C03591=1030.387,347.262,-133.744,171.985,46.375,159.086
C03592=1030.379,347.015,-133.707,171.979,46.373,159.085
C03593=1030.371,346.768,-133.670,171.972,46.372,159.084
C03594=1030.363,346.521,-133.633,171.966,46.372,159.083
C03595=1030.356,346.273,-133.596,171.960,46.371,159.082
C03596=1030.348,346.026,-133.559,171.954,46.370,159.081
C03597=1030.341,345.779,-133.521,171.948,46.368,159.080
C03598=1030.333,345.532,-133.484,171.942,46.367,159.079
C03599=1030.325,345.285,-133.447,171.936,46.366,159.078
C03600=1030.317,345.038,-133.410,171.930,46.365,159.077
C03601=1030.310,344.791,-133.372,171.924,46.364,159.076
C03602=1030.302,344.544,-133.336,171.918,46.363,159.075
C03603=1030.295,344.297,-133.298,171.912,46.362,159.074
C03604=1030.287,344.050,-133.262,171.906,46.361,159.073
C03605=1030.280,343.803,-133.224,171.899,46.360,159.072
C03606=1030.272,343.555,-133.188,171.894,46.359,159.072
C03607=1030.264,343.308,-133.151,171.887,46.358,159.071
C03608=1030.257,343.061,-133.113,171.881,46.357,159.070
C03609=1030.249,342.814,-133.077,171.875,46.356,159.069
C03610=1030.242,342.567,-133.040,171.869,46.355,159.068
C03611=1030.234,342.319,-133.003,171.864,46.354,159.067
C03612=1030.226,342.072,-132.966,171.858,46.353,159.066
C03613=1030.219,341.825,-132.929,171.852,46.352,159.065
C03614=1030.212,341.578,-132.893,171.846,46.351,159.064
C03615=1030.204,341.331,-132.855,171.840,46.350,159.063
C03616=1030.197,341.083,-132.819,171.833,46.349,159.062
C03617=1030.189,340.836,-132.783,171.828,46.349,159.061
C03618=1030.182,340.589,-132.746,171.822,46.347,159.060
C03619=1030.175,340.342,-132.709,171.816,46.347,159.060
C03620=1030.167,340.095,-132.672,171.810,46.346,159.059
C03621=1030.159,339.848,-132.636,171.804,46.345,159.058
C03622=1030.151,339.600,-132.600,171.798,46.344,159.057
C03623=1030.144,339.352,-132.563,171.792,46.343,159.056
C03624=1030.136,339.106,-132.526,171.787,46.343,159.055
C03625=1030.129,338.859,-132.490,171.781,46.341,159.054
C03626=1030.122,338.611,-132.454,171.775,46.341,159.053
C03627=1030.114,338.364,-132.418,171.769,46.340,159.053
C03628=1030.106,338.116,-132.382,171.763,46.339,159.052
C03629=1030.099,337.869,-132.346,171.758,46.338,159.051
C03630=1030.092,337.623,-132.308,171.752,46.338,159.050
C03631=1030.084,337.375,-132.272,171.746,46.337,159.049
C03632=1030.077,337.128,-132.236,171.740,46.336,159.048
C03633=1030.069,336.880,-132.200,171.734,46.336,159.047
C03634=1030.062,336.633,-132.164,171.729,46.335,159.047
C03635=1030.049,336.216,-132.102,171.720,46.334,159.045
C03636=1030.037,335.800,-132.042,171.710,46.332,159.044
C03637=1030.024,335.383,-131.981,171.701,46.331,159.042
C03638=1030.012,334.966,-131.920,171.691,46.330,159.041
C03639=1030.005,334.718,-131.884,171.685,46.330,159.040
C03640=1029.998,334.472,-131.848,171.679,46.328,159.039
C03641=1029.990,334.224,-131.812,171.674,46.328,159.038
C03642=1029.982,333.977,-131.776,171.668,46.327,159.038
C03643=1029.975,333.730,-131.740,171.662,46.326,159.037
C03644=1029.968,333.482,-131.704,171.656,46.326,159.036
C03645=1029.961,333.235,-131.669,171.652,46.326,159.035
C03646=1029.953,332.988,-131.632,171.646,46.325,159.034
C03647=1029.945,332.740,-131.597,171.640,46.325,159.034
C03648=1029.938,332.493,-131.562,171.635,46.324,159.033
C03649=1029.930,332.246,-131.525,171.629,46.323,159.032
C03650=1029.924,331.998,-131.490,171.623,46.323,159.031
C03651=1029.916,331.751,-131.454,171.617,46.322,159.030
C03652=1029.909,331.504,-131.419,171.612,46.321,159.030
C03653=1029.901,331.256,-131.383,171.606,46.321,159.029
C03654=1029.895,331.009,-131.347,171.601,46.321,159.028
C03655=1029.886,330.762,-131.312,171.596,46.320,159.027
C03656=1029.879,330.514,-131.277,171.590,46.319,159.027
C03657=1029.872,330.267,-131.241,171.584,46.319,159.026
C03658=1029.865,330.019,-131.205,171.579,46.319,159.025
C03659=1029.857,329.772,-131.169,171.574,46.318,159.024
C03660=1029.851,329.525,-131.134,171.569,46.317,159.024
C03661=1029.843,329.277,-131.098,171.563,46.317,159.023
C03662=1029.835,329.030,-131.063,171.557,46.317,159.022
C03663=1029.829,328.783,-131.028,171.552,46.316,159.021
C03664=1029.821,328.535,-130.992,171.546,46.315,159.021
C03665=1029.814,328.288,-130.957,171.541,46.316,159.020
C03666=1029.807,328.040,-130.921,171.536,46.315,159.019
C03667=1029.800,327.793,-130.885,171.530,46.314,159.018
C03668=1029.792,327.546,-130.851,171.525,46.314,159.018
C03669=1029.785,327.298,-130.815,171.519,46.313,159.017
C03670=1029.777,327.051,-130.781,171.514,46.313,159.016
C03671=1029.769,326.803,-130.746,171.509,46.313,159.015
C03672=1029.762,326.556,-130.711,171.503,46.313,159.015
C03673=1029.755,326.309,-130.676,171.498,46.313,159.014
C03674=1029.748,326.061,-130.641,171.493,46.312,159.013
C03675=1029.740,325.814,-130.606,171.487,46.312,159.013
C03676=1029.733,325.566,-130.571,171.482,46.311,159.012
C03677=1029.725,325.319,-130.536,171.477,46.311,159.011
C03678=1029.718,325.071,-130.502,171.471,46.311,159.011
C03679=1029.711,324.824,-130.467,171.466,46.310,159.010
C03680=1029.703,324.576,-130.432,171.460,46.310,159.009
C03681=1029.696,324.329,-130.396,171.456,46.310,159.009
C03682=1029.689,324.081,-130.363,171.450,46.310,159.008
C03683=1029.682,323.833,-130.327,171.444,46.310,159.007
C03684=1029.674,323.586,-130.293,171.440,46.310,159.007
C03685=1029.666,323.339,-130.258,171.434,46.310,159.006
C03686=1029.660,323.092,-130.223,171.429,46.309,159.005
C03687=1029.652,322.844,-130.188,171.424,46.309,159.005
C03688=1029.645,322.596,-130.154,171.419,46.309,159.004
C03689=1029.638,322.349,-130.119,171.413,46.309,159.003
C03690=1029.630,322.102,-130.085,171.408,46.308,159.003
C03691=1029.624,321.891,-130.054,171.404,46.308,159.002
C03692=1029.618,321.680,-130.026,171.399,46.308,159.002
C03693=1029.612,321.470,-129.996,171.395,46.308,159.001
C03694=1029.605,321.259,-129.967,171.390,46.308,159.000
C03695=1029.600,321.049,-129.937,171.386,46.307,159.000
C03696=1029.593,320.838,-129.907,171.381,46.307,158.999
C03697=1029.588,320.627,-129.878,171.377,46.307,158.999
C03698=1029.581,320.417,-129.849,171.373,46.307,158.998
C03699=1029.575,320.169,-129.814,171.367,46.307,158.998
C03700=1029.567,319.922,-129.780,171.363,46.306,158.997
C03701=1029.560,319.674,-129.745,171.357,46.306,158.996
C03702=1029.553,319.426,-129.711,171.352,46.306,158.996
C03703=1029.545,319.179,-129.676,171.347,46.306,158.995
C03704=1029.539,318.931,-129.642,171.342,46.306,158.994
C03705=1029.531,318.684,-129.607,171.337,46.306,158.994
C03706=1029.525,318.436,-129.573,171.332,46.306,158.993
C03707=1029.517,318.189,-129.538,171.327,46.306,158.993
C03708=1029.510,317.941,-129.505,171.322,46.306,158.992
C03709=1029.503,317.694,-129.469,171.317,46.305,158.991
C03710=1029.496,317.446,-129.436,171.311,46.305,158.991
C03711=1029.489,317.199,-129.401,171.307,46.305,158.990
C03712=1029.482,316.951,-129.367,171.301,46.305,158.989
C03713=1029.475,316.703,-129.333,171.297,46.305,158.989
C03714=1029.468,316.456,-129.298,171.291,46.305,158.988
C03715=1029.462,316.209,-129.264,171.286,46.305,158.988
C03716=1029.454,315.961,-129.230,171.282,46.305,158.987
C03717=1029.448,315.714,-129.195,171.276,46.305,158.987
C03718=1029.440,315.466,-129.161,171.272,46.305,158.986
C03719=1029.433,315.219,-129.128,171.266,46.305,158.985
C03720=1029.427,314.971,-129.093,171.262,46.305,158.985
C03721=1029.419,314.724,-129.059,171.257,46.305,158.984
C03722=1029.412,314.476,-129.025,171.251,46.305,158.984
C03723=1029.406,314.229,-128.991,171.247,46.305,158.983
C03724=1029.399,313.981,-128.957,171.241,46.305,158.982
C03725=1029.392,313.734,-128.922,171.237,46.305,158.982
C03726=1029.385,313.486,-128.888,171.232,46.305,158.981
C03727=1029.378,313.238,-128.854,171.227,46.305,158.981
C03728=1029.371,312.991,-128.820,171.222,46.305,158.980
C03729=1029.365,312.743,-128.786,171.218,46.305,158.980
C03730=1029.358,312.496,-128.752,171.212,46.305,158.979
C03731=1029.351,312.248,-128.718,171.207,46.305,158.978
C03732=1029.344,312.000,-128.684,171.203,46.305,158.978
C03733=1029.337,311.753,-128.651,171.197,46.305,158.977
C03734=1029.331,311.505,-128.616,171.193,46.305,158.977
C03735=1029.324,311.257,-128.583,171.188,46.305,158.976
C03736=1029.317,311.010,-128.549,171.183,46.306,158.976
C03737=1029.310,310.763,-128.515,171.178,46.305,158.975
C03738=1029.303,310.515,-128.481,171.174,46.306,158.975
C03739=1029.295,310.268,-128.448,171.168,46.306,158.974
C03740=1029.288,310.019,-128.415,171.164,46.306,158.974
C03741=1029.281,309.772,-128.382,171.158,46.306,158.973
C03742=1029.273,309.525,-128.348,171.154,46.307,158.973
C03743=1029.266,309.277,-128.315,171.149,46.306,158.972
C03744=1029.259,309.029,-128.281,171.144,46.307,158.972
C03745=1029.253,308.782,-128.248,171.140,46.307,158.971
C03746=1029.245,308.535,-128.215,171.134,46.307,158.970
C03747=1029.238,308.286,-128.182,171.130,46.308,158.970
C03748=1029.231,308.040,-128.148,171.126,46.308,158.970
C03749=1029.224,307.791,-128.115,171.120,46.308,158.969
C03750=1029.216,307.544,-128.082,171.116,46.309,158.969
C03751=1029.205,307.127,-128.026,171.108,46.309,158.968
C03752=1029.193,306.711,-127.970,171.099,46.309,158.967
C03753=1029.181,306.295,-127.914,171.091,46.310,158.966
C03754=1029.170,305.879,-127.859,171.084,46.311,158.965
C03755=1029.162,305.631,-127.825,171.079,46.311,158.965
C03756=1029.155,305.384,-127.793,171.074,46.312,158.964
C03757=1029.148,305.136,-127.759,171.069,46.311,158.964
C03758=1029.141,304.888,-127.726,171.065,46.312,158.963
C03759=1029.134,304.640,-127.694,171.060,46.312,158.963
C03760=1029.127,304.393,-127.660,171.055,46.313,158.963
C03761=1029.121,304.145,-127.627,171.051,46.313,158.962
C03762=1029.113,303.897,-127.595,171.046,46.313,158.961
C03763=1029.107,303.650,-127.561,171.041,46.314,158.961
C03764=1029.100,303.402,-127.528,171.037,46.314,158.961
C03765=1029.093,303.154,-127.495,171.033,46.314,158.960
C03766=1029.085,302.907,-127.462,171.027,46.315,158.960
C03767=1029.079,302.659,-127.429,171.023,46.316,158.959
C03768=1029.072,302.411,-127.396,171.019,46.316,158.959
C03769=1029.065,302.164,-127.364,171.014,46.316,158.958
C03770=1029.058,301.916,-127.330,171.009,46.316,158.958
C03771=1029.052,301.668,-127.298,171.004,46.317,158.957
C03772=1029.044,301.420,-127.265,171.000,46.317,158.957
C03773=1029.038,301.173,-127.232,170.996,46.318,158.957
C03774=1029.031,300.925,-127.199,170.990,46.318,158.956
C03775=1029.025,300.677,-127.166,170.986,46.319,158.956
C03776=1029.017,300.430,-127.133,170.982,46.319,158.955
C03777=1029.010,300.182,-127.100,170.977,46.319,158.955
C03778=1029.004,299.934,-127.068,170.973,46.320,158.954
C03779=1028.996,299.686,-127.035,170.968,46.320,158.954
C03780=1028.990,299.439,-127.002,170.963,46.321,158.954
C03781=1028.983,299.191,-126.969,170.959,46.321,158.953
C03782=1028.976,298.943,-126.937,170.955,46.322,158.953
C03783=1028.970,298.696,-126.904,170.950,46.322,158.952
C03784=1028.963,298.447,-126.871,170.945,46.323,158.952
C03785=1028.956,298.200,-126.839,170.941,46.323,158.951
C03786=1028.950,297.953,-126.806,170.936,46.323,158.951
C03787=1028.943,297.704,-126.773,170.932,46.324,158.951
C03788=1028.936,297.457,-126.741,170.928,46.324,158.950
C03789=1028.930,297.209,-126.708,170.922,46.325,158.950
C03790=1028.923,296.962,-126.676,170.918,46.325,158.949
C03791=1028.916,296.714,-126.643,170.914,46.326,158.949
C03792=1028.909,296.466,-126.610,170.909,46.326,158.948
C03793=1028.903,296.219,-126.578,170.905,46.327,158.948
C03794=1028.896,295.970,-126.546,170.901,46.328,158.948
C03795=1028.889,295.722,-126.513,170.897,46.328,158.947
C03796=1028.883,295.475,-126.480,170.891,46.329,158.947
C03797=1028.876,295.228,-126.448,170.887,46.329,158.946
C03798=1028.870,294.980,-126.416,170.883,46.329,158.946
C03799=1028.863,294.732,-126.382,170.878,46.330,158.946
C03800=1028.856,294.484,-126.351,170.874,46.331,158.945
C03801=1028.850,294.236,-126.318,170.870,46.331,158.945
C03802=1028.843,293.989,-126.286,170.866,46.332,158.945
C03803=1028.836,293.740,-126.254,170.860,46.332,158.944
C03804=1028.829,293.493,-126.222,170.856,46.333,158.944
C03805=1028.822,293.245,-126.189,170.852,46.334,158.943
C03806=1028.816,292.997,-126.157,170.848,46.334,158.943
C03807=1028.804,292.598,-126.106,170.840,46.335,158.942
C03808=1028.794,292.199,-126.054,170.834,46.336,158.942
C03809=1028.783,291.800,-126.002,170.827,46.337,158.941
C03810=1028.772,291.400,-125.951,170.820,46.339,158.941
C03811=1028.765,291.153,-125.919,170.815,46.339,158.940
C03812=1028.759,290.905,-125.887,170.811,46.340,158.940
C03813=1028.752,290.657,-125.855,170.807,46.341,158.940
C03814=1028.745,290.409,-125.824,170.803,46.341,158.939
C03815=1028.738,290.161,-125.792,170.799,46.342,158.939
C03816=1028.731,289.914,-125.760,170.793,46.343,158.939
C03817=1028.725,289.665,-125.728,170.789,46.344,158.938
C03818=1028.718,289.417,-125.696,170.785,46.344,158.938
C03819=1028.711,289.170,-125.664,170.781,46.345,158.938
C03820=1028.704,288.922,-125.633,170.777,46.346,158.938
C03821=1028.697,288.674,-125.601,170.772,46.347,158.937
C03822=1028.690,288.427,-125.569,170.768,46.348,158.937
C03823=1028.684,288.179,-125.537,170.764,46.348,158.936
C03824=1028.677,287.930,-125.505,170.759,46.350,158.936
C03825=1028.670,287.682,-125.474,170.755,46.350,158.936
C03826=1028.664,287.434,-125.442,170.751,46.351,158.935
C03827=1028.657,287.187,-125.410,170.747,46.352,158.935
C03828=1028.650,286.939,-125.379,170.742,46.352,158.935
C03829=1028.643,286.691,-125.347,170.738,46.353,158.935
C03830=1028.636,286.443,-125.316,170.734,46.354,158.934
C03831=1028.630,286.196,-125.284,170.730,46.355,158.934
C03832=1028.624,285.947,-125.252,170.726,46.356,158.934
C03833=1028.617,285.699,-125.221,170.722,46.357,158.933
C03834=1028.609,285.452,-125.190,170.717,46.357,158.933
C03835=1028.603,285.204,-125.159,170.712,46.359,158.933
C03836=1028.596,284.956,-125.127,170.708,46.360,158.932
C03837=1028.589,284.708,-125.096,170.704,46.361,158.932
C03838=1028.583,284.460,-125.064,170.700,46.361,158.932
C03839=1028.576,284.212,-125.033,170.696,46.362,158.932
C03840=1028.569,283.964,-125.001,170.692,46.363,158.931
C03841=1028.562,283.716,-124.970,170.688,46.364,158.931
C03842=1028.556,283.469,-124.939,170.684,46.365,158.931
C03843=1028.548,283.221,-124.908,170.680,46.366,158.931
C03844=1028.542,282.973,-124.876,170.676,46.367,158.930
C03845=1028.535,282.725,-124.846,170.671,46.368,158.930
C03846=1028.528,282.477,-124.814,170.667,46.369,158.930
C03847=1028.522,282.229,-124.783,170.663,46.370,158.929
C03848=1028.515,281.981,-124.751,170.658,46.371,158.929
C03849=1028.508,281.733,-124.720,170.654,46.372,158.929
C03850=1028.501,281.485,-124.688,170.650,46.373,158.929
C03851=1028.495,281.237,-124.658,170.646,46.373,158.928
C03852=1028.488,280.989,-124.627,170.642,46.374,158.928
C03853=1028.481,280.741,-124.595,170.638,46.375,158.928
C03854=1028.475,280.494,-124.564,170.634,46.376,158.927
C03855=1028.468,280.245,-124.534,170.630,46.377,158.927
C03856=1028.462,279.997,-124.502,170.626,46.378,158.927
C03857=1028.455,279.749,-124.471,170.622,46.379,158.927
C03858=1028.448,279.501,-124.440,170.618,46.381,158.926
C03859=1028.442,279.253,-124.409,170.614,46.382,158.926
C03860=1028.434,279.005,-124.378,170.610,46.383,158.926
C03861=1028.428,278.758,-124.347,170.606,46.384,158.926
C03862=1028.422,278.510,-124.316,170.601,46.385,158.925
C03863=1028.411,278.122,-124.267,170.595,46.386,158.925
C03864=1028.401,277.736,-124.219,170.589,46.388,158.925
C03865=1028.391,277.349,-124.171,170.582,46.389,158.924
C03866=1028.380,276.962,-124.122,170.576,46.391,158.924
C03867=1028.373,276.713,-124.092,170.572,46.392,158.924
C03868=1028.367,276.466,-124.062,170.568,46.393,158.923
C03869=1028.360,276.218,-124.031,170.564,46.394,158.923
C03870=1028.354,275.969,-124.000,170.560,46.396,158.923
C03871=1028.346,275.722,-123.969,170.556,46.397,158.923
C03872=1028.340,275.474,-123.939,170.552,46.398,158.923
C03873=1028.333,275.226,-123.908,170.548,46.399,158.922
C03874=1028.327,274.978,-123.877,170.544,46.400,158.922
C03875=1028.320,274.729,-123.846,170.540,46.401,158.922
C03876=1028.313,274.482,-123.815,170.536,46.403,158.922
C03877=1028.307,274.234,-123.785,170.532,46.404,158.922
C03878=1028.300,273.985,-123.754,170.528,46.405,158.921
C03879=1028.293,273.737,-123.724,170.524,46.406,158.921
C03880=1028.287,273.490,-123.693,170.520,46.407,158.921
C03881=1028.280,273.242,-123.663,170.516,46.408,158.921
C03882=1028.274,272.993,-123.632,170.512,46.409,158.921
C03883=1028.266,272.745,-123.602,170.508,46.410,158.920
C03884=1028.260,272.498,-123.571,170.504,46.411,158.920
C03885=1028.254,272.249,-123.540,170.501,46.413,158.920
C03886=1028.247,272.001,-123.510,170.497,46.414,158.920
C03887=1028.241,271.753,-123.480,170.493,46.415,158.919
C03888=1028.234,271.505,-123.450,170.489,46.417,158.919
C03889=1028.227,271.257,-123.418,170.485,46.418,158.919
C03890=1028.220,271.009,-123.389,170.481,46.419,158.919
C03891=1028.214,270.761,-123.358,170.477,46.421,158.919
C03892=1028.207,270.513,-123.328,170.474,46.421,158.919
C03893=1028.201,270.265,-123.298,170.470,46.422,158.918
C03894=1028.194,270.017,-123.267,170.466,46.424,158.918
C03895=1028.187,269.768,-123.237,170.462,46.425,158.918
C03896=1028.181,269.521,-123.207,170.458,46.427,158.918
C03897=1028.174,269.272,-123.177,170.454,46.428,158.918
C03898=1028.167,269.024,-123.146,170.450,46.429,158.917
C03899=1028.161,268.776,-123.116,170.446,46.430,158.917
C03900=1028.154,268.528,-123.086,170.442,46.431,158.917
C03901=1028.148,268.280,-123.056,170.439,46.433,158.917
C03902=1028.141,268.032,-123.026,170.435,46.434,158.917
C03903=1028.133,267.784,-122.996,170.431,46.436,158.917
C03904=1028.128,267.536,-122.965,170.427,46.437,158.916
C03905=1028.121,267.288,-122.935,170.423,46.438,158.916
C03906=1028.114,267.040,-122.905,170.419,46.440,158.916
C03907=1028.108,266.791,-122.875,170.415,46.441,158.916
C03908=1028.101,266.544,-122.846,170.411,46.442,158.916
C03909=1028.094,266.296,-122.816,170.407,46.444,158.916
C03910=1028.088,266.047,-122.785,170.403,46.445,158.916
C03911=1028.081,265.799,-122.755,170.401,46.446,158.916
C03912=1028.074,265.551,-122.726,170.397,46.447,158.915
C03913=1028.068,265.303,-122.696,170.393,46.449,158.915
C03914=1028.061,265.055,-122.665,170.389,46.451,158.915
C03915=1028.055,264.807,-122.635,170.385,46.452,158.915
C03916=1028.048,264.558,-122.606,170.381,46.453,158.915
C03917=1028.041,264.311,-122.576,170.377,46.454,158.915
C03918=1028.034,264.063,-122.546,170.374,46.456,158.914
C03919=1028.024,263.680,-122.500,170.368,46.458,158.914
C03920=1028.014,263.298,-122.454,170.362,46.460,158.914
C03921=1028.004,262.915,-122.408,170.356,46.463,158.914
C03922=1027.994,262.533,-122.363,170.350,46.465,158.914
C03923=1027.987,262.285,-122.332,170.347,46.466,158.914
C03924=1027.981,262.037,-122.303,170.343,46.467,158.913
C03925=1027.974,261.788,-122.273,170.339,46.469,158.913
C03926=1027.968,261.540,-122.244,170.335,46.471,158.913
C03927=1027.961,261.293,-122.214,170.331,46.472,158.913
C03928=1027.954,261.044,-122.184,170.328,46.473,158.913
C03929=1027.948,260.796,-122.155,170.325,46.475,158.913
C03930=1027.941,260.548,-122.126,170.321,46.477,158.913
C03931=1027.934,260.300,-122.096,170.317,46.478,158.913
C03932=1027.927,260.051,-122.066,170.313,46.480,158.913
C03933=1027.921,259.804,-122.037,170.310,46.482,158.912
C03934=1027.913,259.555,-122.008,170.306,46.483,158.912
C03935=1027.907,259.307,-121.979,170.302,46.484,158.912
C03936=1027.900,259.059,-121.949,170.298,46.486,158.912
C03937=1027.894,258.811,-121.920,170.294,46.488,158.912
C03938=1027.887,258.563,-121.891,170.291,46.489,158.912
C03939=1027.880,258.314,-121.862,170.287,46.491,158.912
C03940=1027.873,258.067,-121.832,170.283,46.493,158.912
C03941=1027.866,257.818,-121.803,170.279,46.494,158.912
C03942=1027.860,257.570,-121.774,170.277,46.496,158.912
C03943=1027.853,257.321,-121.744,170.273,46.497,158.912
C03944=1027.846,257.074,-121.715,170.269,46.499,158.912
C03945=1027.840,256.825,-121.686,170.265,46.501,158.911
C03946=1027.833,256.577,-121.657,170.262,46.502,158.911
C03947=1027.827,256.328,-121.627,170.258,46.504,158.911
C03948=1027.820,256.081,-121.599,170.254,46.506,158.911
C03949=1027.812,255.832,-121.569,170.250,46.507,158.911
C03950=1027.806,255.584,-121.540,170.247,46.509,158.911
C03951=1027.799,255.335,-121.510,170.243,46.511,158.911
C03952=1027.793,255.087,-121.481,170.240,46.512,158.911
C03953=1027.786,254.839,-121.453,170.236,46.514,158.911
C03954=1027.779,254.591,-121.424,170.233,46.516,158.911
C03955=1027.773,254.342,-121.395,170.229,46.517,158.911
C03956=1027.767,254.094,-121.365,170.225,46.519,158.911
C03957=1027.760,253.847,-121.337,170.221,46.521,158.911
C03958=1027.753,253.598,-121.307,170.217,46.522,158.910
C03959=1027.746,253.350,-121.278,170.214,46.524,158.910
C03960=1027.740,253.102,-121.249,170.211,46.525,158.910
C03961=1027.733,252.853,-121.219,170.207,46.527,158.910
C03962=1027.726,252.605,-121.191,170.203,46.529,158.910
C03963=1027.720,252.357,-121.162,170.200,46.530,158.910
C03964=1027.714,252.109,-121.133,170.196,46.532,158.910
C03965=1027.707,251.860,-121.103,170.192,46.534,158.910
C03966=1027.700,251.612,-121.075,170.188,46.535,158.910
C03967=1027.694,251.364,-121.046,170.186,46.537,158.910
C03968=1027.687,251.116,-121.017,170.182,46.539,158.910
C03969=1027.681,250.867,-120.988,170.179,46.541,158.910
C03970=1027.674,250.620,-120.959,170.175,46.542,158.910
C03971=1027.668,250.371,-120.931,170.171,46.544,158.910
C03972=1027.661,250.123,-120.902,170.167,46.546,158.910
C03973=1027.655,249.875,-120.873,170.164,46.547,158.910
C03974=1027.648,249.626,-120.844,170.161,46.549,158.909
C03975=1027.638,249.242,-120.799,170.155,46.552,158.909
C03976=1027.628,248.859,-120.754,170.150,46.555,158.909
C03977=1027.618,248.475,-120.710,170.144,46.557,158.909
C03978=1027.608,248.091,-120.665,170.139,46.560,158.909
C03979=1027.601,247.843,-120.636,170.135,46.562,158.909
C03980=1027.595,247.594,-120.608,170.132,46.563,158.909
C03981=1027.589,247.346,-120.579,170.129,46.565,158.909
C03982=1027.583,247.098,-120.550,170.125,46.567,158.909
C03983=1027.576,246.850,-120.522,170.121,46.569,158.909
C03984=1027.569,246.601,-120.492,170.118,46.571,158.909
C03985=1027.563,246.353,-120.464,170.115,46.572,158.909
C03986=1027.557,246.105,-120.435,170.111,46.574,158.909
C03987=1027.550,245.857,-120.406,170.107,46.575,158.909
C03988=1027.543,245.609,-120.377,170.104,46.578,158.909
C03989=1027.537,245.360,-120.349,170.101,46.579,158.909
C03990=1027.531,245.112,-120.320,170.097,46.581,158.909
C03991=1027.524,244.864,-120.291,170.094,46.583,158.909
C03992=1027.518,244.615,-120.263,170.090,46.585,158.909
C03993=1027.512,244.367,-120.234,170.086,46.587,158.909
C03994=1027.505,244.119,-120.206,170.084,46.588,158.909
C03995=1027.499,243.870,-120.177,170.080,46.590,158.909
C03996=1027.492,243.623,-120.149,170.076,46.592,158.909
C03997=1027.486,243.374,-120.121,170.073,46.594,158.909
C03998=1027.479,243.125,-120.092,170.069,46.596,158.909
C03999=1027.473,242.877,-120.063,170.066,46.597,158.909
C04000=1027.466,242.629,-120.035,170.063,46.599,158.909
C04001=1027.460,242.380,-120.007,170.059,46.601,158.909
C04002=1027.453,242.132,-119.978,170.055,46.603,158.909
C04003=1027.447,241.883,-119.950,170.053,46.605,158.909
C04004=1027.440,241.636,-119.921,170.049,46.607,158.909
C04005=1027.434,241.387,-119.893,170.046,46.609,158.909
C04006=1027.427,241.139,-119.865,170.042,46.611,158.909
C04007=1027.420,240.891,-119.837,170.038,46.613,158.909
C04008=1027.414,240.642,-119.808,170.036,46.615,158.909
C04009=1027.407,240.394,-119.780,170.032,46.616,158.909
C04010=1027.401,240.145,-119.752,170.029,46.619,158.909
C04011=1027.394,239.897,-119.723,170.025,46.620,158.909
C04012=1027.388,239.649,-119.696,170.021,46.623,158.909
C04013=1027.382,239.400,-119.667,170.019,46.624,158.909
C04014=1027.375,239.152,-119.639,170.015,46.626,158.909
C04015=1027.368,238.904,-119.611,170.011,46.628,158.909
C04016=1027.361,238.656,-119.583,170.008,46.630,158.909
C04017=1027.355,238.407,-119.556,170.005,46.633,158.909
C04018=1027.348,238.159,-119.527,170.002,46.634,158.909
C04019=1027.342,237.911,-119.499,169.998,46.636,158.909
C04020=1027.335,237.662,-119.471,169.995,46.638,158.909
C04021=1027.328,237.414,-119.443,169.991,46.641,158.909
C04022=1027.322,237.165,-119.416,169.988,46.643,158.909
C04023=1027.315,236.917,-119.387,169.985,46.644,158.909
C04024=1027.309,236.669,-119.359,169.981,46.647,158.909
C04025=1027.302,236.420,-119.331,169.978,46.649,158.909
C04026=1027.295,236.172,-119.304,169.974,46.651,158.909
C04027=1027.289,235.924,-119.276,169.971,46.653,158.909
C04028=1027.283,235.676,-119.248,169.968,46.655,158.909
C04029=1027.276,235.427,-119.221,169.965,46.657,158.909
C04030=1027.270,235.178,-119.192,169.961,46.659,158.909
C04031=1027.259,234.789,-119.149,169.956,46.663,158.909
C04032=1027.249,234.398,-119.104,169.950,46.665,158.909
C04033=1027.239,234.009,-119.061,169.945,46.669,158.910
C04034=1027.229,233.619,-119.018,169.940,46.672,158.910
C04035=1027.222,233.370,-118.990,169.937,46.674,158.910
C04036=1027.215,233.122,-118.962,169.934,46.676,158.910
C04037=1027.209,232.873,-118.934,169.930,46.678,158.910
C04038=1027.202,232.625,-118.907,169.927,46.681,158.910
C04039=1027.196,232.377,-118.879,169.924,46.682,158.910
C04040=1027.189,232.129,-118.852,169.921,46.685,158.910
C04041=1027.183,231.880,-118.824,169.917,46.687,158.910
C04042=1027.177,231.631,-118.795,169.914,46.689,158.910
C04043=1027.170,231.383,-118.768,169.911,46.691,158.910
C04044=1027.163,231.135,-118.740,169.908,46.693,158.910
C04045=1027.157,230.887,-118.713,169.904,46.695,158.910
C04046=1027.150,230.638,-118.685,169.901,46.698,158.910
C04047=1027.144,230.390,-118.657,169.898,46.700,158.911
C04048=1027.137,230.141,-118.630,169.894,46.701,158.910
C04049=1027.131,229.892,-118.602,169.891,46.704,158.911
C04050=1027.124,229.644,-118.575,169.888,46.706,158.911
C04051=1027.118,229.396,-118.547,169.885,46.708,158.911
C04052=1027.111,229.148,-118.520,169.882,46.711,158.911
C04053=1027.105,228.899,-118.492,169.878,46.713,158.911
C04054=1027.098,228.650,-118.465,169.875,46.715,158.911
C04055=1027.092,228.402,-118.437,169.872,46.717,158.911
C04056=1027.085,228.154,-118.410,169.869,46.719,158.911
C04057=1027.079,227.906,-118.382,169.865,46.721,158.911
C04058=1027.072,227.657,-118.356,169.862,46.724,158.911
C04059=1027.065,227.408,-118.328,169.859,46.726,158.911
C04060=1027.059,227.161,-118.301,169.856,46.728,158.911
C04061=1027.053,226.912,-118.274,169.852,46.730,158.912
C04062=1027.046,226.663,-118.246,169.849,46.733,158.912
C04063=1027.038,226.415,-118.219,169.846,46.735,158.912
C04064=1027.033,226.167,-118.192,169.843,46.737,158.912
C04065=1027.026,225.918,-118.164,169.839,46.740,158.912
C04066=1027.020,225.669,-118.137,169.836,46.742,158.912
C04067=1027.012,225.421,-118.110,169.832,46.744,158.912
C04068=1027.006,225.173,-118.082,169.830,46.746,158.912
C04069=1027.000,224.924,-118.056,169.827,46.749,158.912
C04070=1026.992,224.676,-118.029,169.823,46.751,158.912
C04071=1026.986,224.427,-118.002,169.820,46.753,158.912
C04072=1026.980,224.179,-117.974,169.817,46.755,158.913
C04073=1026.974,223.930,-117.947,169.814,46.758,158.913
C04074=1026.966,223.682,-117.920,169.811,46.761,158.913
C04075=1026.960,223.433,-117.893,169.807,46.763,158.913
C04076=1026.954,223.185,-117.866,169.805,46.765,158.913
C04077=1026.947,222.937,-117.839,169.801,46.768,158.913
C04078=1026.940,222.688,-117.812,169.798,46.770,158.913
C04079=1026.934,222.440,-117.785,169.794,46.772,158.913
C04080=1026.927,222.191,-117.757,169.792,46.774,158.914
C04081=1026.920,221.943,-117.731,169.788,46.777,158.914
C04082=1026.914,221.695,-117.703,169.785,46.779,158.914
C04083=1026.908,221.446,-117.676,169.782,46.781,158.914
C04084=1026.901,221.197,-117.650,169.779,46.784,158.914
C04085=1026.895,220.949,-117.623,169.776,46.786,158.914
C04086=1026.888,220.700,-117.596,169.772,46.789,158.914
C04087=1026.877,220.303,-117.552,169.767,46.792,158.914
C04088=1026.868,219.905,-117.509,169.762,46.796,158.915
C04089=1026.857,219.508,-117.466,169.758,46.800,158.915
C04090=1026.847,219.110,-117.423,169.753,46.803,158.915
C04091=1026.840,218.861,-117.396,169.750,46.806,158.915
C04092=1026.833,218.613,-117.369,169.746,46.809,158.915
C04093=1026.826,218.365,-117.343,169.743,46.811,158.915
C04094=1026.820,218.116,-117.316,169.741,46.814,158.916
C04095=1026.813,217.868,-117.289,169.737,46.816,158.916
C04096=1026.807,217.619,-117.262,169.734,46.818,158.916
C04097=1026.800,217.370,-117.236,169.730,46.821,158.916
C04098=1026.794,217.122,-117.209,169.728,46.823,158.916
C04099=1026.787,216.873,-117.183,169.725,46.826,158.916
C04100=1026.780,216.625,-117.157,169.721,46.828,158.916
C04101=1026.774,216.377,-117.129,169.718,46.831,158.917
C04102=1026.767,216.128,-117.103,169.716,46.833,158.917
C04103=1026.761,215.880,-117.076,169.712,46.836,158.917
C04104=1026.754,215.631,-117.050,169.709,46.839,158.917
C04105=1026.748,215.382,-117.023,169.706,46.841,158.917
C04106=1026.741,215.134,-116.996,169.703,46.843,158.917
C04107=1026.734,214.886,-116.970,169.700,46.846,158.918
C04108=1026.728,214.637,-116.943,169.697,46.848,158.918
C04109=1026.721,214.388,-116.917,169.693,46.851,158.918
C04110=1026.715,214.140,-116.890,169.691,46.853,158.918
C04111=1026.708,213.891,-116.863,169.687,46.856,158.918
C04112=1026.701,213.643,-116.837,169.684,46.859,158.918
C04113=1026.695,213.394,-116.810,169.682,46.861,158.919
C04114=1026.688,213.146,-116.784,169.678,46.863,158.919
C04115=1026.682,212.897,-116.757,169.675,46.866,158.919
C04116=1026.675,212.649,-116.731,169.672,46.869,158.919
C04117=1026.669,212.400,-116.704,169.669,46.871,158.919
C04118=1026.662,212.152,-116.678,169.666,46.874,158.919
C04119=1026.655,211.903,-116.652,169.663,46.876,158.919
C04120=1026.650,211.655,-116.625,169.661,46.879,158.920
C04121=1026.642,211.406,-116.598,169.657,46.881,158.920
C04122=1026.637,211.158,-116.572,169.654,46.884,158.920
C04123=1026.630,210.909,-116.545,169.651,46.886,158.920
C04124=1026.623,210.661,-116.519,169.648,46.889,158.920
C04125=1026.617,210.412,-116.492,169.645,46.892,158.921
C04126=1026.610,210.163,-116.467,169.641,46.894,158.921
C04127=1026.604,209.915,-116.441,169.639,46.897,158.921
C04128=1026.597,209.666,-116.415,169.636,46.899,158.921
C04129=1026.590,209.418,-116.388,169.633,46.902,158.921
C04130=1026.584,209.169,-116.361,169.629,46.905,158.921
C04131=1026.577,208.921,-116.335,169.627,46.907,158.922
C04132=1026.570,208.673,-116.309,169.624,46.910,158.922
C04133=1026.564,208.424,-116.284,169.620,46.913,158.922
C04134=1026.558,208.175,-116.257,169.618,46.915,158.922
C04135=1026.551,207.927,-116.231,169.615,46.918,158.922
C04136=1026.544,207.678,-116.204,169.612,46.921,158.923
C04137=1026.538,207.429,-116.179,169.608,46.923,158.923
C04138=1026.531,207.181,-116.153,169.606,46.926,158.923
C04139=1026.524,206.933,-116.126,169.603,46.928,158.923
C04140=1026.518,206.685,-116.100,169.599,46.931,158.923
C04141=1026.512,206.435,-116.074,169.597,46.934,158.924
C04142=1026.505,206.187,-116.048,169.594,46.936,158.924
C04143=1026.494,205.793,-116.006,169.589,46.941,158.924
C04144=1026.484,205.399,-115.966,169.584,46.945,158.924
C04145=1026.474,205.006,-115.924,169.580,46.950,158.925
C04146=1026.463,204.611,-115.884,169.575,46.954,158.925
C04147=1026.439,203.573,-115.781,169.186,46.851,158.855
C04148=1026.432,203.324,-115.756,169.182,46.855,158.856
C04149=1026.427,203.076,-115.732,169.178,46.858,158.856
C04150=1026.421,202.827,-115.708,169.174,46.862,158.856
C04151=1026.415,202.578,-115.683,169.170,46.865,158.856
C04152=1026.409,202.329,-115.658,169.166,46.869,158.857
C04153=1026.403,202.081,-115.634,169.162,46.873,158.857
C04154=1026.397,201.832,-115.610,169.158,46.876,158.857
C04155=1026.392,201.583,-115.585,169.155,46.880,158.857
C04156=1026.386,201.334,-115.561,169.151,46.883,158.858
C04157=1026.381,201.086,-115.536,169.147,46.887,158.858
C04158=1026.375,200.838,-115.512,169.143,46.890,158.858
C04159=1026.369,200.588,-115.488,169.139,46.894,158.858
C04160=1026.363,200.340,-115.463,169.135,46.897,158.859
C04161=1026.357,200.090,-115.439,169.131,46.901,158.859
C04162=1026.351,199.842,-115.415,169.127,46.904,158.859
C04163=1026.345,199.593,-115.390,169.124,46.908,158.859
C04164=1026.339,199.345,-115.367,169.119,46.912,158.860
C04165=1026.334,199.095,-115.342,169.116,46.915,158.860
C04166=1026.328,198.847,-115.318,169.112,46.919,158.860
C04167=1026.321,198.598,-115.294,169.107,46.923,158.860
C04168=1026.316,198.350,-115.270,169.104,46.927,158.861
C04169=1026.309,198.101,-115.246,169.100,46.931,158.861
C04170=1026.304,197.851,-115.223,169.095,46.934,158.861
C04171=1026.298,197.603,-115.199,169.092,46.938,158.862
C04172=1026.292,197.354,-115.174,169.089,46.942,158.862
C04173=1026.286,197.105,-115.151,169.084,46.945,158.862
C04174=1026.279,196.856,-115.127,169.081,46.949,158.862
C04175=1026.274,196.608,-115.102,169.077,46.953,158.863
C04176=1026.268,196.360,-115.079,169.072,46.956,158.863
C04177=1026.262,196.110,-115.055,169.069,46.960,158.863
C04178=1026.256,195.861,-115.031,169.065,46.964,158.864
C04179=1026.251,195.613,-115.007,169.062,46.967,158.864
C04180=1026.244,195.364,-114.983,169.058,46.971,158.864
C04181=1026.238,195.116,-114.959,169.054,46.975,158.864
C04182=1026.233,194.866,-114.936,169.050,46.978,158.865
C04183=1026.227,194.617,-114.912,169.046,46.982,158.865
C04184=1026.221,194.369,-114.887,169.042,46.986,158.865
C04185=1026.215,194.121,-114.864,169.039,46.989,158.865
C04186=1026.209,193.871,-114.840,169.035,46.993,158.866
C04187=1026.204,193.622,-114.816,169.031,46.997,158.866
C04188=1026.198,193.374,-114.792,169.027,47.000,158.866
C04189=1026.192,193.124,-114.769,169.023,47.004,158.867
C04190=1026.186,192.876,-114.745,169.019,47.008,158.867
C04191=1026.181,192.627,-114.721,169.016,47.012,158.867
C04192=1026.175,192.379,-114.697,169.012,47.015,158.867
C04193=1026.168,192.129,-114.674,169.008,47.019,158.868
C04194=1026.163,191.881,-114.649,169.004,47.023,158.868
C04195=1026.157,191.632,-114.626,169.001,47.026,158.868
C04196=1026.152,191.383,-114.602,168.997,47.030,158.869
C04197=1026.145,191.134,-114.578,168.993,47.034,158.869
C04198=1026.140,190.885,-114.555,168.989,47.038,158.869
C04199=1026.134,190.637,-114.531,168.986,47.041,158.870
C04200=1026.129,190.388,-114.508,168.982,47.045,158.870
C04201=1026.123,190.139,-114.483,168.978,47.049,158.870
C04202=1026.117,189.890,-114.460,168.974,47.053,158.871
C04203=1026.111,189.642,-114.437,168.971,47.056,158.871
C04204=1026.106,189.393,-114.413,168.967,47.060,158.871
C04205=1026.100,189.144,-114.390,168.963,47.064,158.871
C04206=1026.094,188.895,-114.365,168.960,47.068,158.872
C04207=1026.088,188.646,-114.342,168.956,47.071,158.872
C04208=1026.083,188.410,-114.319,168.952,47.075,158.872
C04209=1026.078,188.174,-114.297,168.949,47.078,158.872
C04210=1026.072,187.938,-114.275,168.945,47.082,158.873
C04211=1026.066,187.702,-114.253,168.943,47.086,158.873
C04212=1026.061,187.466,-114.230,168.938,47.089,158.873
C04213=1026.056,187.231,-114.208,168.935,47.093,158.874
C04214=1026.051,186.994,-114.185,168.931,47.096,158.874
C04215=1026.046,186.758,-114.163,168.928,47.100,158.874
C04216=1026.040,186.509,-114.140,168.925,47.104,158.875
C04217=1026.034,186.260,-114.117,168.921,47.107,158.875
C04218=1026.028,186.011,-114.092,168.917,47.111,158.875
C04219=1026.022,185.762,-114.069,168.914,47.115,158.875
C04220=1026.017,185.514,-114.045,168.911,47.118,158.876
C04221=1026.011,185.265,-114.022,168.907,47.122,158.876
C04222=1026.006,185.016,-113.999,168.903,47.126,158.876
C04223=1026.000,184.767,-113.975,168.900,47.129,158.877
C04224=1025.995,184.518,-113.952,168.896,47.133,158.877
C04225=1025.989,184.269,-113.929,168.892,47.137,158.877
C04226=1025.984,184.021,-113.905,168.889,47.140,158.878
C04227=1025.978,183.772,-113.882,168.885,47.144,158.878
C04228=1025.973,183.523,-113.858,168.881,47.148,158.878
C04229=1025.967,183.274,-113.835,168.878,47.152,158.879
C04230=1025.961,183.026,-113.812,168.874,47.155,158.879
C04231=1025.956,182.776,-113.788,168.871,47.159,158.879
C04232=1025.950,182.527,-113.765,168.867,47.163,158.879
C04233=1025.944,182.278,-113.742,168.863,47.167,158.880
C04234=1025.938,182.029,-113.719,168.860,47.171,158.880
C04235=1025.932,181.781,-113.696,168.857,47.175,158.881
C04236=1025.926,181.532,-113.673,168.853,47.179,158.881
C04237=1025.920,181.283,-113.650,168.849,47.183,158.881
C04238=1025.914,181.035,-113.628,168.845,47.187,158.882
C04239=1025.908,180.785,-113.605,168.842,47.191,158.882
C04240=1025.902,180.536,-113.582,168.839,47.195,158.882
C04241=1025.897,180.287,-113.559,168.835,47.199,158.883
C04242=1025.890,180.039,-113.537,168.832,47.203,158.883
C04243=1025.885,179.790,-113.514,168.828,47.207,158.883
C04244=1025.877,179.481,-113.485,168.823,47.212,158.884
C04245=1025.870,179.173,-113.457,168.819,47.217,158.884
C04246=1025.862,178.865,-113.429,168.815,47.222,158.885
C04247=1025.855,178.556,-113.401,168.811,47.227,158.885
C04248=1025.849,178.308,-113.378,168.807,47.231,158.886
C04249=1025.844,178.059,-113.355,168.803,47.235,158.886
C04250=1025.837,177.810,-113.333,168.800,47.239,158.886
C04251=1025.832,177.561,-113.311,168.796,47.243,158.887
C04252=1025.826,177.312,-113.288,168.793,47.247,158.887
C04253=1025.820,177.063,-113.265,168.790,47.250,158.887
C04254=1025.814,176.814,-113.242,168.786,47.255,158.888
C04255=1025.808,176.565,-113.219,168.782,47.259,158.888
C04256=1025.802,176.316,-113.196,168.779,47.263,158.888
C04257=1025.797,176.067,-113.174,168.776,47.267,158.889
C04258=1025.791,175.818,-113.152,168.772,47.271,158.889
C04259=1025.785,175.569,-113.129,168.769,47.275,158.890
C04260=1025.779,175.320,-113.106,168.765,47.279,158.890
C04261=1025.773,175.072,-113.084,168.761,47.283,158.890
C04262=1025.767,174.822,-113.061,168.758,47.287,158.891
C04263=1025.761,174.573,-113.038,168.755,47.291,158.891
C04264=1025.756,174.325,-113.016,168.752,47.295,158.891
C04265=1025.750,174.076,-112.994,168.748,47.299,158.892
C04266=1025.744,173.827,-112.971,168.744,47.303,158.892
C04267=1025.739,173.578,-112.948,168.741,47.306,158.892
C04268=1025.733,173.329,-112.925,168.737,47.310,158.893
C04269=1025.727,173.080,-112.904,168.734,47.315,158.893
C04270=1025.721,172.831,-112.881,168.731,47.319,158.894
C04271=1025.715,172.582,-112.858,168.727,47.323,158.894
C04272=1025.709,172.299,-112.833,168.723,47.328,158.894
C04273=1025.702,172.017,-112.807,168.720,47.332,158.895
C04274=1025.696,171.733,-112.781,168.716,47.336,158.895
C04275=1025.689,171.450,-112.756,168.711,47.341,158.896
C04276=1025.684,171.201,-112.733,168.709,47.345,158.896
C04277=1025.678,170.952,-112.712,168.705,47.349,158.896
C04278=1025.672,170.703,-112.689,168.702,47.353,158.897
C04279=1025.667,170.454,-112.666,168.698,47.357,158.897
C04280=1025.660,170.205,-112.644,168.695,47.361,158.898
C04281=1025.655,169.956,-112.621,168.692,47.365,158.898
C04282=1025.649,169.707,-112.599,168.689,47.369,158.898
C04283=1025.644,169.458,-112.576,168.685,47.373,158.899
C04284=1025.638,169.210,-112.554,168.681,47.377,158.899
C04285=1025.632,168.961,-112.532,168.678,47.381,158.899
C04286=1025.627,168.712,-112.509,168.674,47.385,158.900
C04287=1025.620,168.462,-112.487,168.672,47.389,158.900
C04288=1025.615,168.214,-112.465,168.668,47.393,158.900
C04289=1025.610,167.965,-112.443,168.665,47.397,158.901
C04290=1025.604,167.716,-112.420,168.661,47.401,158.901
C04291=1025.598,167.467,-112.398,168.658,47.405,158.902
C04292=1025.593,167.218,-112.376,168.654,47.409,158.902
C04293=1025.587,166.969,-112.353,168.652,47.413,158.902
C04294=1025.581,166.720,-112.331,168.648,47.417,158.903
C04295=1025.576,166.471,-112.309,168.645,47.421,158.903
C04296=1025.570,166.223,-112.286,168.641,47.425,158.903
C04297=1025.564,165.973,-112.264,168.638,47.429,158.904
C04298=1025.559,165.724,-112.242,168.635,47.433,158.904
C04299=1025.554,165.476,-112.220,168.632,47.436,158.904
C04300=1025.548,165.227,-112.198,168.628,47.441,158.905
C04301=1025.542,164.978,-112.175,168.625,47.445,158.905
C04302=1025.537,164.729,-112.153,168.621,47.449,158.906
C04303=1025.532,164.479,-112.131,168.619,47.453,158.906
C04304=1025.525,164.231,-112.109,168.616,47.456,158.906
C04305=1025.520,163.982,-112.087,168.612,47.460,158.907
C04306=1025.515,163.733,-112.064,168.609,47.465,158.907
C04307=1025.508,163.484,-112.042,168.606,47.469,158.908
C04308=1025.504,163.235,-112.020,168.603,47.473,158.908
C04309=1025.498,162.986,-111.997,168.599,47.477,158.908
C04310=1025.492,162.737,-111.976,168.596,47.480,158.909
C04311=1025.487,162.488,-111.954,168.592,47.484,158.909
C04312=1025.481,162.239,-111.931,168.589,47.488,158.909
C04313=1025.475,161.990,-111.909,168.587,47.493,158.910
C04314=1025.470,161.741,-111.887,168.583,47.497,158.910
C04315=1025.464,161.492,-111.864,168.580,47.500,158.911
C04316=1025.459,161.244,-111.843,168.576,47.504,158.911
C04317=1025.453,160.994,-111.821,168.573,47.508,158.911
C04318=1025.448,160.745,-111.799,168.570,47.512,158.912
C04319=1025.442,160.497,-111.777,168.567,47.517,158.912
C04320=1025.437,160.247,-111.755,168.564,47.520,158.912
C04321=1025.432,159.998,-111.733,168.560,47.525,158.913
C04322=1025.426,159.749,-111.711,168.557,47.528,158.913
C04323=1025.421,159.501,-111.688,168.555,47.532,158.914
C04324=1025.415,159.252,-111.666,168.551,47.536,158.914
C04325=1025.409,159.002,-111.645,168.548,47.541,158.914
C04326=1025.403,158.754,-111.623,168.544,47.545,158.915
C04327=1025.397,158.505,-111.602,168.541,47.548,158.915
C04328=1025.392,158.255,-111.579,168.538,47.553,158.916
C04329=1025.386,158.007,-111.558,168.535,47.557,158.916
C04330=1025.380,157.757,-111.537,168.532,47.562,158.916
C04331=1025.375,157.509,-111.515,168.529,47.565,158.917
C04332=1025.369,157.259,-111.493,168.525,47.569,158.917
C04333=1025.363,157.010,-111.471,168.522,47.574,158.918
C04334=1025.357,156.762,-111.450,168.519,47.578,158.918
C04335=1025.351,156.512,-111.429,168.516,47.582,158.919
C04336=1025.346,156.229,-111.404,168.512,47.587,158.919
C04337=1025.339,155.945,-111.380,168.509,47.592,158.919
C04338=1025.332,155.662,-111.355,168.505,47.596,158.920
C04339=1025.326,155.378,-111.330,168.502,47.601,158.920
C04340=1025.320,155.129,-111.309,168.498,47.605,158.921
C04341=1025.314,154.880,-111.287,168.495,47.609,158.921
C04342=1025.309,154.631,-111.266,168.493,47.613,158.922
C04343=1025.302,154.382,-111.244,168.489,47.617,158.922
C04344=1025.298,154.133,-111.223,168.486,47.621,158.922
C04345=1025.291,153.884,-111.201,168.482,47.626,158.923
C04346=1025.286,153.636,-111.180,168.479,47.630,158.923
C04347=1025.280,153.386,-111.159,168.477,47.634,158.924
C04348=1025.274,153.137,-111.137,168.473,47.638,158.924
C04349=1025.268,152.888,-111.116,168.471,47.643,158.925
C04350=1025.263,152.639,-111.094,168.467,47.647,158.925
C04351=1025.257,152.390,-111.072,168.464,47.651,158.925
C04352=1025.252,152.141,-111.052,168.460,47.655,158.926
C04353=1025.246,151.892,-111.030,168.458,47.659,158.926
C04354=1025.240,151.643,-111.009,168.455,47.664,158.927
C04355=1025.234,151.394,-110.987,168.451,47.668,158.927
C04356=1025.229,151.145,-110.967,168.449,47.672,158.928
C04357=1025.223,150.896,-110.945,168.445,47.676,158.928
C04358=1025.217,150.647,-110.924,168.442,47.681,158.928
C04359=1025.211,150.397,-110.903,168.439,47.684,158.929
C04360=1025.206,150.149,-110.882,168.436,47.688,158.929
C04361=1025.200,149.900,-110.860,168.433,47.693,158.930
C04362=1025.194,149.651,-110.839,168.429,47.697,158.930
C04363=1025.188,149.401,-110.818,168.427,47.701,158.930
C04364=1025.183,149.153,-110.797,168.424,47.705,158.931
C04365=1025.177,148.904,-110.775,168.420,47.710,158.931
C04366=1025.171,148.655,-110.754,168.418,47.714,158.932
C04367=1025.166,148.406,-110.733,168.414,47.718,158.932
C04368=1025.160,148.156,-110.712,168.411,47.722,158.933
C04369=1025.154,147.908,-110.691,168.409,47.727,158.933
C04370=1025.148,147.659,-110.669,168.405,47.731,158.933
C04371=1025.143,147.409,-110.649,168.402,47.735,158.934
C04372=1025.137,147.161,-110.627,168.399,47.739,158.934
C04373=1025.131,146.911,-110.607,168.396,47.743,158.935
C04374=1025.126,146.663,-110.585,168.393,47.748,158.935
C04375=1025.120,146.413,-110.564,168.389,47.752,158.935
C04376=1025.114,146.164,-110.543,168.387,47.756,158.936
C04377=1025.109,145.915,-110.522,168.384,47.760,158.936
C04378=1025.103,145.666,-110.501,168.380,47.765,158.937
C04379=1025.098,145.417,-110.480,168.378,47.769,158.937
C04380=1025.091,145.168,-110.459,168.375,47.773,158.938
C04381=1025.086,144.919,-110.439,168.372,47.778,158.938
C04382=1025.080,144.670,-110.417,168.369,47.781,158.939
C04383=1025.074,144.420,-110.397,168.365,47.786,158.939
C04384=1025.069,144.172,-110.375,168.362,47.790,158.939
C04385=1025.063,143.923,-110.355,168.360,47.794,158.940
C04386=1025.057,143.673,-110.334,168.356,47.799,158.940
C04387=1025.051,143.425,-110.313,168.354,47.803,158.941
C04388=1025.045,143.175,-110.292,168.351,47.807,158.941
C04389=1025.040,142.926,-110.271,168.347,47.812,158.942
C04390=1025.034,142.678,-110.251,168.345,47.816,158.942
C04391=1025.028,142.428,-110.230,168.341,47.820,158.943
C04392=1025.022,142.179,-110.209,168.338,47.825,158.943
C04393=1025.017,141.930,-110.188,168.336,47.828,158.943
C04394=1025.011,141.680,-110.167,168.332,47.833,158.944
C04395=1025.005,141.432,-110.147,168.329,47.837,158.944
C04396=1025.000,141.183,-110.126,168.327,47.841,158.945
C04397=1024.994,140.934,-110.106,168.323,47.846,158.945
C04398=1024.988,140.685,-110.084,168.320,47.850,158.946
C04399=1024.982,140.436,-110.064,168.318,47.855,158.946
C04400=1024.975,140.152,-110.040,168.314,47.859,158.947
C04401=1024.970,139.868,-110.017,168.311,47.864,158.947
C04402=1024.963,139.584,-109.993,168.307,47.869,158.948
C04403=1024.957,139.300,-109.969,168.304,47.874,158.948
C04404=1024.951,139.051,-109.948,168.301,47.878,158.949
C04405=1024.945,138.802,-109.928,168.297,47.882,158.949
C04406=1024.939,138.553,-109.907,168.295,47.887,158.950
C04407=1024.934,138.304,-109.887,168.292,47.890,158.950
C04408=1024.928,138.054,-109.866,168.289,47.895,158.950
C04409=1024.922,137.806,-109.846,168.286,47.900,158.951
C04410=1024.917,137.556,-109.825,168.283,47.903,158.951
C04411=1024.910,137.308,-109.804,168.280,47.908,158.952
C04412=1024.905,137.058,-109.784,168.277,47.912,158.952
C04413=1024.900,136.809,-109.763,168.274,47.917,158.953
C04414=1024.894,136.560,-109.743,168.272,47.921,158.953
C04415=1024.888,136.311,-109.722,168.268,47.925,158.954
C04416=1024.882,136.062,-109.702,168.266,47.930,158.954
C04417=1024.877,135.813,-109.682,168.263,47.934,158.955
C04418=1024.871,135.564,-109.662,168.259,47.938,158.955
C04419=1024.865,135.315,-109.641,168.257,47.943,158.955
C04420=1024.859,135.065,-109.621,168.254,47.947,158.956
C04421=1024.853,134.817,-109.600,168.250,47.951,158.956
C04422=1024.847,134.568,-109.580,168.248,47.956,158.957
C04423=1024.842,134.319,-109.559,168.245,47.960,158.957
C04424=1024.835,134.069,-109.539,168.242,47.964,158.958
C04425=1024.830,133.820,-109.518,168.239,47.969,158.958
C04426=1024.824,133.571,-109.498,168.236,47.973,158.959
C04427=1024.819,133.322,-109.478,168.233,47.977,158.959
C04428=1024.814,133.073,-109.457,168.230,47.982,158.960
C04429=1024.807,132.824,-109.437,168.228,47.986,158.960
C04430=1024.802,132.574,-109.416,168.225,47.990,158.961
C04431=1024.796,132.326,-109.396,168.221,47.994,158.961
C04432=1024.790,132.077,-109.376,168.219,47.999,158.961
C04433=1024.785,131.827,-109.356,168.216,48.003,158.962
C04434=1024.779,131.578,-109.336,168.212,48.008,158.962
C04435=1024.773,131.328,-109.316,168.210,48.012,158.963
C04436=1024.768,131.079,-109.295,168.207,48.017,158.963
C04437=1024.762,130.831,-109.275,168.205,48.020,158.964
C04438=1024.756,130.581,-109.255,168.201,48.025,158.964
C04439=1024.750,130.333,-109.235,168.198,48.029,158.964
C04440=1024.744,130.084,-109.215,168.196,48.033,158.965
C04441=1024.739,129.835,-109.194,168.192,48.038,158.965
C04442=1024.733,129.585,-109.174,168.190,48.043,158.966
C04443=1024.727,129.336,-109.154,168.187,48.047,158.966
C04444=1024.721,129.087,-109.135,168.184,48.051,158.967
C04445=1024.715,128.838,-109.115,168.181,48.056,158.967
C04446=1024.709,128.589,-109.095,168.179,48.060,158.968
C04447=1024.704,128.340,-109.075,168.175,48.065,158.968
C04448=1024.697,128.090,-109.054,168.172,48.069,158.969
C04449=1024.691,127.841,-109.034,168.170,48.074,158.969
C04450=1024.686,127.592,-109.015,168.166,48.078,158.970
C04451=1024.680,127.343,-108.995,168.164,48.083,158.970
C04452=1024.674,127.094,-108.975,168.161,48.087,158.971
C04453=1024.669,126.844,-108.955,168.159,48.091,158.971
C04454=1024.663,126.596,-108.936,168.155,48.096,158.972
C04455=1024.657,126.347,-108.916,168.153,48.100,158.972
C04456=1024.651,126.097,-108.896,168.150,48.104,158.973
C04457=1024.644,125.848,-108.876,168.146,48.109,158.973
C04458=1024.638,125.599,-108.856,168.144,48.114,158.974
C04459=1024.634,125.349,-108.836,168.141,48.118,158.974
C04460=1024.628,125.100,-108.816,168.138,48.122,158.974
C04461=1024.622,124.852,-108.796,168.135,48.127,158.975
C04462=1024.616,124.602,-108.777,168.133,48.131,158.976
C04463=1024.610,124.353,-108.757,168.130,48.136,158.976
C04464=1024.603,124.070,-108.735,168.127,48.141,158.977
C04465=1024.597,123.785,-108.711,168.123,48.146,158.977
C04466=1024.590,123.501,-108.689,168.120,48.151,158.978
C04467=1024.584,123.218,-108.667,168.116,48.156,158.978
C04468=1024.578,122.968,-108.648,168.114,48.160,158.979
C04469=1024.572,122.720,-108.628,168.111,48.165,158.979
C04470=1024.566,122.471,-108.608,168.108,48.170,158.980
C04471=1024.561,122.221,-108.588,168.105,48.173,158.980
C04472=1024.555,121.972,-108.568,168.103,48.178,158.981
C04473=1024.549,121.722,-108.548,168.100,48.182,158.981
C04474=1024.543,121.473,-108.528,168.096,48.187,158.981
C04475=1024.537,121.224,-108.509,168.094,48.191,158.982
C04476=1024.531,120.975,-108.489,168.091,48.196,158.982
C04477=1024.526,120.726,-108.470,168.089,48.200,158.983
C04478=1024.520,120.476,-108.449,168.085,48.204,158.983
C04479=1024.515,120.227,-108.430,168.083,48.209,158.984
C04480=1024.509,119.978,-108.410,168.080,48.213,158.984
C04481=1024.503,119.729,-108.391,168.077,48.217,158.985
C04482=1024.497,119.481,-108.371,168.074,48.222,158.985
C04483=1024.492,119.231,-108.352,168.072,48.227,158.986
C04484=1024.486,118.982,-108.332,168.069,48.230,158.986
C04485=1024.481,118.733,-108.312,168.066,48.235,158.987
C04486=1024.475,118.484,-108.292,168.064,48.239,158.987
C04487=1024.469,118.234,-108.273,168.060,48.244,158.987
C04488=1024.463,117.986,-108.253,168.058,48.248,158.988
C04489=1024.457,117.736,-108.234,168.055,48.253,158.989
C04490=1024.452,117.487,-108.215,168.053,48.257,158.989
C04491=1024.446,117.238,-108.195,168.050,48.261,158.989
C04492=1024.440,116.988,-108.175,168.046,48.266,158.990
C04493=1024.435,116.739,-108.155,168.044,48.270,158.990
C04494=1024.429,116.490,-108.136,168.041,48.274,158.991
C04495=1024.423,116.240,-108.116,168.039,48.279,158.991
C04496=1024.418,115.992,-108.096,168.036,48.283,158.992
C04497=1024.412,115.742,-108.077,168.032,48.287,158.992
C04498=1024.406,115.494,-108.058,168.030,48.292,158.993
C04499=1024.401,115.245,-108.038,168.027,48.296,158.993
C04500=1024.395,114.995,-108.019,168.025,48.300,158.994
C04501=1024.390,114.746,-107.998,168.022,48.305,158.994
C04502=1024.384,114.497,-107.979,168.019,48.309,158.995
C04503=1024.378,114.247,-107.960,168.016,48.314,158.995
C04504=1024.372,113.998,-107.940,168.013,48.318,158.996
C04505=1024.367,113.749,-107.921,168.011,48.322,158.996
C04506=1024.362,113.500,-107.902,168.008,48.327,158.996
C04507=1024.356,113.251,-107.882,168.006,48.331,158.997
C04508=1024.350,113.002,-107.863,168.003,48.335,158.997
C04509=1024.345,112.752,-107.843,168.001,48.340,158.998
C04510=1024.339,112.503,-107.824,167.997,48.344,158.998
C04511=1024.333,112.254,-107.804,167.994,48.348,158.999
C04512=1024.327,112.005,-107.785,167.992,48.353,158.999
C04513=1024.321,111.755,-107.766,167.989,48.357,159.000
C04514=1024.316,111.506,-107.747,167.986,48.362,159.000
C04515=1024.310,111.257,-107.728,167.983,48.366,159.001
C04516=1024.305,111.008,-107.708,167.981,48.371,159.001
C04517=1024.298,110.759,-107.689,167.978,48.375,159.002
C04518=1024.292,110.510,-107.670,167.976,48.380,159.002
C04519=1024.287,110.261,-107.651,167.972,48.384,159.002
C04520=1024.281,110.011,-107.631,167.969,48.388,159.003
C04521=1024.275,109.762,-107.612,167.967,48.393,159.004
C04522=1024.269,109.513,-107.594,167.965,48.398,159.004
C04523=1024.264,109.264,-107.575,167.962,48.402,159.005
C04524=1024.258,109.014,-107.555,167.958,48.406,159.005
C04525=1024.252,108.765,-107.537,167.956,48.411,159.005
C04526=1024.246,108.516,-107.517,167.953,48.415,159.006
C04527=1024.240,108.266,-107.498,167.951,48.420,159.007
C04528=1024.233,107.982,-107.477,167.948,48.425,159.007
C04529=1024.227,107.699,-107.455,167.944,48.430,159.008
C04530=1024.221,107.414,-107.433,167.941,48.435,159.008
C04531=1024.214,107.131,-107.412,167.938,48.441,159.009
C04532=1024.208,106.881,-107.393,167.935,48.445,159.009
C04533=1024.202,106.632,-107.374,167.933,48.450,159.010
C04534=1024.196,106.383,-107.355,167.930,48.454,159.010
C04535=1024.191,106.134,-107.336,167.928,48.458,159.011
C04536=1024.184,105.885,-107.318,167.924,48.463,159.011
C04537=1024.179,105.635,-107.298,167.922,48.468,159.012
C04538=1024.173,105.386,-107.279,167.919,48.472,159.012
C04539=1024.167,105.137,-107.261,167.917,48.476,159.013
C04540=1024.161,104.888,-107.242,167.914,48.481,159.013
C04541=1024.156,104.639,-107.222,167.911,48.485,159.014
C04542=1024.150,104.389,-107.204,167.908,48.490,159.014
C04543=1024.144,104.140,-107.185,167.906,48.495,159.015
C04544=1024.139,103.891,-107.166,167.903,48.498,159.015
C04545=1024.132,103.642,-107.148,167.901,48.503,159.016
C04546=1024.127,103.392,-107.128,167.898,48.508,159.016
C04547=1024.122,103.143,-107.109,167.895,48.512,159.017
C04548=1024.115,102.894,-107.091,167.892,48.516,159.017
C04549=1024.109,102.645,-107.072,167.889,48.521,159.017
C04550=1024.104,102.395,-107.053,167.887,48.525,159.018
C04551=1024.098,102.146,-107.035,167.885,48.530,159.019
C04552=1024.093,101.897,-107.016,167.882,48.535,159.019
C04553=1024.086,101.648,-106.997,167.878,48.539,159.019
C04554=1024.081,101.399,-106.978,167.876,48.543,159.020
C04555=1024.075,101.150,-106.959,167.873,48.548,159.020
C04556=1024.069,100.900,-106.941,167.871,48.552,159.021
C04557=1024.064,100.650,-106.922,167.868,48.556,159.021
C04558=1024.058,100.402,-106.903,167.866,48.561,159.022
C04559=1024.052,100.153,-106.884,167.863,48.566,159.022
C04560=1024.046,99.903,-106.865,167.860,48.570,159.023
C04561=1024.042,99.654,-106.847,167.857,48.574,159.023
C04562=1024.035,99.405,-106.828,167.855,48.579,159.024
C04563=1024.029,99.156,-106.809,167.852,48.583,159.024
C04564=1024.024,98.906,-106.791,167.850,48.588,159.025
C04565=1024.017,98.657,-106.773,167.846,48.593,159.025
C04566=1024.011,98.408,-106.754,167.844,48.597,159.026
C04567=1024.006,98.158,-106.735,167.841,48.601,159.026
C04568=1024.000,97.909,-106.717,167.839,48.606,159.027
C04569=1023.994,97.659,-106.699,167.836,48.610,159.027
C04570=1023.988,97.410,-106.680,167.833,48.615,159.028
C04571=1023.982,97.162,-106.662,167.830,48.620,159.028
C04572=1023.977,96.912,-106.643,167.828,48.625,159.029
C04573=1023.970,96.663,-106.624,167.826,48.629,159.029
C04574=1023.965,96.414,-106.607,167.823,48.633,159.030
C04575=1023.959,96.164,-106.588,167.819,48.638,159.030
C04576=1023.953,95.915,-106.569,167.817,48.642,159.031
C04577=1023.947,95.666,-106.551,167.815,48.647,159.031
C04578=1023.942,95.417,-106.532,167.812,48.652,159.032
C04579=1023.935,95.167,-106.514,167.810,48.656,159.032
C04580=1023.930,94.918,-106.496,167.807,48.660,159.033
C04581=1023.924,94.668,-106.477,167.803,48.665,159.033
C04582=1023.918,94.420,-106.459,167.801,48.670,159.034
C04583=1023.912,94.170,-106.441,167.799,48.674,159.034
C04584=1023.907,93.921,-106.422,167.796,48.679,159.035
C04585=1023.901,93.672,-106.404,167.793,48.683,159.035
C04586=1023.895,93.423,-106.386,167.791,48.687,159.036
C04587=1023.889,93.173,-106.367,167.788,48.692,159.036
C04588=1023.883,92.924,-106.349,167.785,48.697,159.036
C04589=1023.877,92.674,-106.331,167.783,48.701,159.037
C04590=1023.872,92.426,-106.312,167.780,48.705,159.037
C04591=1023.866,92.176,-106.294,167.778,48.710,159.038
C04592=1023.859,91.892,-106.273,167.774,48.715,159.039
C04593=1023.853,91.609,-106.253,167.771,48.720,159.039
C04594=1023.847,91.324,-106.231,167.769,48.726,159.040
C04595=1023.840,91.040,-106.211,167.765,48.730,159.040
C04596=1023.834,90.791,-106.192,167.763,48.735,159.041
C04597=1023.829,90.541,-106.174,167.761,48.740,159.041
C04598=1023.823,90.293,-106.156,167.758,48.744,159.042
C04599=1023.817,90.043,-106.138,167.754,48.748,159.042
C04600=1023.812,89.794,-106.119,167.752,48.753,159.043
C04601=1023.805,89.545,-106.101,167.750,48.758,159.043
C04602=1023.799,89.295,-106.083,167.747,48.761,159.043
C04603=1023.794,89.046,-106.065,167.744,48.766,159.044
C04604=1023.787,88.797,-106.047,167.742,48.771,159.044
C04605=1023.782,88.548,-106.029,167.739,48.776,159.045
C04606=1023.776,88.298,-106.011,167.736,48.780,159.045
C04607=1023.770,88.050,-105.993,167.734,48.785,159.046
C04608=1023.764,87.800,-105.975,167.731,48.789,159.047
C04609=1023.758,87.550,-105.957,167.729,48.794,159.047
C04610=1023.752,87.301,-105.939,167.725,48.799,159.048
C04611=1023.746,87.051,-105.922,167.723,48.803,159.048
C04612=1023.741,86.803,-105.903,167.720,48.807,159.048
C04613=1023.735,86.553,-105.885,167.718,48.812,159.049
C04614=1023.729,86.304,-105.867,167.716,48.817,159.049
C04615=1023.723,86.054,-105.849,167.713,48.821,159.050
C04616=1023.717,85.806,-105.831,167.710,48.826,159.050
C04617=1023.711,85.556,-105.813,167.707,48.831,159.051
C04618=1023.706,85.307,-105.795,167.705,48.835,159.052
C04619=1023.700,85.057,-105.777,167.702,48.840,159.052
C04620=1023.694,84.808,-105.760,167.700,48.844,159.052
C04621=1023.688,84.558,-105.742,167.696,48.849,159.053
C04622=1023.682,84.310,-105.724,167.694,48.853,159.053
C04623=1023.676,84.060,-105.706,167.691,48.858,159.054
C04624=1023.671,83.811,-105.688,167.689,48.863,159.054
C04625=1023.664,83.561,-105.670,167.687,48.867,159.055
C04626=1023.659,83.312,-105.653,167.684,48.871,159.055
C04627=1023.653,83.063,-105.635,167.681,48.876,159.056
C04628=1023.647,82.814,-105.617,167.678,48.881,159.056
C04629=1023.641,82.564,-105.599,167.676,48.885,159.057
C04630=1023.635,82.316,-105.581,167.673,48.890,159.057
C04631=1023.630,82.066,-105.563,167.671,48.894,159.058
C04632=1023.624,81.817,-105.545,167.668,48.898,159.058
C04633=1023.618,81.568,-105.528,167.666,48.903,159.059
C04634=1023.612,81.318,-105.510,167.663,48.908,159.059
C04635=1023.607,81.069,-105.492,167.660,48.913,159.060
C04636=1023.600,80.819,-105.474,167.657,48.917,159.060
C04637=1023.595,80.570,-105.457,167.655,48.921,159.061
C04638=1023.589,80.320,-105.439,167.652,48.926,159.061
C04639=1023.583,80.071,-105.421,167.650,48.930,159.062
C04640=1023.578,79.822,-105.404,167.648,48.935,159.062
C04641=1023.572,79.573,-105.386,167.645,48.940,159.063
C04642=1023.566,79.324,-105.368,167.641,48.944,159.063
C04643=1023.560,79.074,-105.350,167.639,48.948,159.064
C04644=1023.554,78.825,-105.333,167.637,48.953,159.064
C04645=1023.549,78.576,-105.315,167.634,48.958,159.065
C04646=1023.543,78.326,-105.297,167.631,48.962,159.065
C04647=1023.537,78.077,-105.280,167.629,48.966,159.066
C04648=1023.532,77.828,-105.262,167.627,48.971,159.066
C04649=1023.526,77.578,-105.244,167.624,48.975,159.067
C04650=1023.520,77.329,-105.227,167.622,48.979,159.067
C04651=1023.514,77.079,-105.209,167.618,48.984,159.067
C04652=1023.508,76.831,-105.192,167.616,48.989,159.068
C04653=1023.502,76.582,-105.174,167.613,48.994,159.068
C04654=1023.496,76.332,-105.156,167.611,48.998,159.069
C04655=1023.491,76.083,-105.139,167.609,49.003,159.069
C04656=1023.483,75.799,-105.119,167.605,49.008,159.070
C04657=1023.477,75.515,-105.099,167.602,49.013,159.071
C04658=1023.470,75.230,-105.079,167.600,49.018,159.071
C04659=1023.464,74.947,-105.059,167.597,49.024,159.072
C04660=1023.458,74.697,-105.042,167.594,49.028,159.072
C04661=1023.451,74.448,-105.025,167.591,49.033,159.073
C04662=1023.446,74.198,-105.008,167.588,49.037,159.073
C04663=1023.441,73.949,-104.990,167.586,49.042,159.074
C04664=1023.434,73.700,-104.972,167.583,49.046,159.074
C04665=1023.428,73.451,-104.955,167.581,49.051,159.075
C04666=1023.423,73.202,-104.938,167.578,49.056,159.075
C04667=1023.417,72.951,-104.920,167.576,49.060,159.076
C04668=1023.411,72.703,-104.903,167.572,49.064,159.076
C04669=1023.405,72.454,-104.886,167.570,49.069,159.076
C04670=1023.399,72.204,-104.868,167.568,49.074,159.077
C04671=1023.394,71.954,-104.851,167.565,49.078,159.077
C04672=1023.387,71.706,-104.834,167.563,49.083,159.078
C04673=1023.381,71.456,-104.816,167.560,49.088,159.079
C04674=1023.376,71.206,-104.799,167.558,49.092,159.079
C04675=1023.370,70.957,-104.782,167.554,49.097,159.079
C04676=1023.364,70.708,-104.765,167.552,49.101,159.080
C04677=1023.358,70.459,-104.747,167.549,49.106,159.080
C04678=1023.352,70.209,-104.731,167.547,49.110,159.081
C04679=1023.347,69.960,-104.713,167.544,49.114,159.081
C04680=1023.341,69.711,-104.695,167.542,49.119,159.082
C04681=1023.335,69.461,-104.679,167.540,49.124,159.082
C04682=1023.329,69.212,-104.661,167.536,49.129,159.083
C04683=1023.324,68.963,-104.644,167.534,49.133,159.083
C04684=1023.317,68.713,-104.627,167.531,49.137,159.084
C04685=1023.312,68.464,-104.610,167.529,49.142,159.084
C04686=1023.306,68.214,-104.593,167.526,49.147,159.085
C04687=1023.300,67.966,-104.576,167.524,49.151,159.085
C04688=1023.294,67.716,-104.558,167.521,49.156,159.086
C04689=1023.288,67.467,-104.542,167.518,49.161,159.086
C04690=1023.283,67.217,-104.524,167.515,49.165,159.087
C04691=1023.276,66.967,-104.507,167.513,49.169,159.087
C04692=1023.270,66.718,-104.490,167.511,49.174,159.088
C04693=1023.265,66.469,-104.474,167.508,49.179,159.088
C04694=1023.259,66.220,-104.456,167.506,49.183,159.089
C04695=1023.253,65.971,-104.440,167.503,49.188,159.089
C04696=1023.247,65.721,-104.422,167.500,49.192,159.089
C04697=1023.241,65.472,-104.406,167.497,49.197,159.090
C04698=1023.235,65.223,-104.388,167.495,49.201,159.090
C04699=1023.229,64.973,-104.372,167.493,49.206,159.091
C04700=1023.223,64.723,-104.354,167.490,49.211,159.092
C04701=1023.217,64.474,-104.338,167.487,49.216,159.092
C04702=1023.212,64.225,-104.320,167.484,49.220,159.092
C04703=1023.206,63.976,-104.304,167.482,49.224,159.093
C04704=1023.201,63.726,-104.287,167.479,49.229,159.093
C04705=1023.194,63.477,-104.270,167.477,49.234,159.094
C04706=1023.189,63.227,-104.253,167.475,49.238,159.094
C04707=1023.182,62.978,-104.236,167.471,49.243,159.095
C04708=1023.176,62.729,-104.219,167.469,49.248,159.095
C04709=1023.170,62.479,-104.203,167.467,49.253,159.096
C04710=1023.165,62.229,-104.186,167.464,49.257,159.096
C04711=1023.158,61.980,-104.169,167.462,49.262,159.097
C04712=1023.152,61.731,-104.153,167.458,49.267,159.097
C04713=1023.147,61.482,-104.136,167.456,49.272,159.098
C04714=1023.140,61.232,-104.119,167.453,49.275,159.098
C04715=1023.134,60.983,-104.103,167.451,49.280,159.099
C04716=1023.129,60.733,-104.086,167.448,49.285,159.099
C04717=1023.123,60.484,-104.070,167.445,49.290,159.100
C04718=1023.116,60.235,-104.053,167.443,49.294,159.100
C04719=1023.110,59.985,-104.036,167.441,49.299,159.101
C04720=1023.103,59.701,-104.018,167.437,49.305,159.101
C04721=1023.097,59.417,-103.999,167.434,49.310,159.102
C04722=1023.090,59.133,-103.980,167.431,49.315,159.102
C04723=1023.083,58.848,-103.961,167.429,49.321,159.103
C04724=1023.077,58.599,-103.944,167.426,49.326,159.104
C04725=1023.071,58.350,-103.928,167.423,49.330,159.104
C04726=1023.065,58.101,-103.911,167.421,49.334,159.104
C04727=1023.059,57.852,-103.895,167.418,49.339,159.105
C04728=1023.054,57.602,-103.878,167.415,49.344,159.105
C04729=1023.048,57.353,-103.862,167.412,49.349,159.106
C04730=1023.042,57.103,-103.845,167.410,49.353,159.106
C04731=1023.035,56.853,-103.829,167.408,49.358,159.107
C04732=1023.029,56.604,-103.812,167.405,49.363,159.108
C04733=1023.023,56.355,-103.796,167.403,49.367,159.108
C04734=1023.018,56.105,-103.779,167.400,49.372,159.108
C04735=1023.012,55.856,-103.763,167.397,49.376,159.109
C04736=1023.006,55.607,-103.746,167.395,49.381,159.109
C04737=1023.000,55.357,-103.730,167.392,49.386,159.110
C04738=1022.994,55.108,-103.714,167.390,49.390,159.110
C04739=1022.988,54.859,-103.697,167.386,49.395,159.111
C04740=1022.982,54.610,-103.680,167.384,49.400,159.111
C04741=1022.976,54.360,-103.664,167.381,49.404,159.112
C04742=1022.970,54.110,-103.647,167.379,49.409,159.112
C04743=1022.964,53.861,-103.631,167.377,49.413,159.113
C04744=1022.958,53.612,-103.615,167.374,49.418,159.113
C04745=1022.952,53.362,-103.598,167.371,49.423,159.114
C04746=1022.946,53.113,-103.582,167.369,49.428,159.114
C04747=1022.941,52.863,-103.565,167.366,49.432,159.115
C04748=1022.935,52.614,-103.549,167.364,49.436,159.115
C04749=1022.929,52.364,-103.533,167.361,49.441,159.116
C04750=1022.923,52.115,-103.516,167.359,49.446,159.116
C04751=1022.917,51.866,-103.500,167.356,49.451,159.117
C04752=1022.911,51.616,-103.484,167.353,49.455,159.117
C04753=1022.905,51.367,-103.468,167.350,49.459,159.117
C04754=1022.900,51.117,-103.451,167.348,49.464,159.118
C04755=1022.894,50.868,-103.435,167.346,49.469,159.118
C04756=1022.888,50.619,-103.418,167.343,49.473,159.119
C04757=1022.882,50.369,-103.402,167.340,49.478,159.119
C04758=1022.876,50.120,-103.386,167.337,49.482,159.120
C04759=1022.870,49.871,-103.370,167.335,49.487,159.120
C04760=1022.864,49.621,-103.353,167.332,49.491,159.121
C04761=1022.859,49.372,-103.336,167.330,49.496,159.121
C04762=1022.853,49.122,-103.320,167.328,49.500,159.122
C04763=1022.847,48.873,-103.304,167.325,49.505,159.122
C04764=1022.841,48.624,-103.288,167.322,49.509,159.122
C04765=1022.835,48.374,-103.271,167.319,49.514,159.123
C04766=1022.829,48.125,-103.255,167.317,49.519,159.123
C04767=1022.823,47.876,-103.239,167.314,49.523,159.124
C04768=1022.817,47.626,-103.223,167.312,49.527,159.124
C04769=1022.812,47.377,-103.206,167.309,49.532,159.125
C04770=1022.806,47.127,-103.190,167.307,49.537,159.125
C04771=1022.800,46.878,-103.173,167.303,49.541,159.126
C04772=1022.795,46.629,-103.157,167.301,49.546,159.126
C04773=1022.789,46.379,-103.142,167.299,49.550,159.127
C04774=1022.783,46.130,-103.126,167.296,49.554,159.127
C04775=1022.777,45.881,-103.109,167.294,49.559,159.128
C04776=1022.772,45.631,-103.092,167.291,49.564,159.128
C04777=1022.766,45.382,-103.076,167.289,49.568,159.128
C04778=1022.760,45.132,-103.060,167.286,49.573,159.129
C04779=1022.754,44.883,-103.044,167.284,49.577,159.129
C04780=1022.749,44.633,-103.028,167.280,49.582,159.130
C04781=1022.743,44.384,-103.012,167.278,49.586,159.130
C04782=1022.737,44.134,-102.996,167.276,49.591,159.131
C04783=1022.731,43.886,-102.980,167.273,49.595,159.131
C04784=1022.724,43.601,-102.961,167.269,49.600,159.131
C04785=1022.718,43.316,-102.943,167.268,49.605,159.132
C04786=1022.712,43.032,-102.924,167.264,49.610,159.133
C04787=1022.705,42.747,-102.906,167.261,49.615,159.133
C04788=1022.699,42.498,-102.889,167.258,49.620,159.134
C04789=1022.694,42.249,-102.874,167.256,49.625,159.134
C04790=1022.688,41.999,-102.858,167.253,49.629,159.134
C04791=1022.682,41.750,-102.842,167.251,49.633,159.135
C04792=1022.676,41.500,-102.827,167.249,49.638,159.135
C04793=1022.670,41.251,-102.810,167.245,49.643,159.136
C04794=1022.664,41.002,-102.794,167.243,49.648,159.136
C04795=1022.658,40.752,-102.779,167.240,49.652,159.137
C04796=1022.652,40.502,-102.762,167.238,49.657,159.137
C04797=1022.647,40.254,-102.747,167.236,49.661,159.138
C04798=1022.641,40.004,-102.732,167.232,49.666,159.138
C04799=1022.635,39.755,-102.715,167.230,49.670,159.139
C04800=1022.629,39.505,-102.700,167.227,49.675,159.139
C04801=1022.623,39.255,-102.684,167.225,49.680,159.140
C04802=1022.617,39.006,-102.667,167.222,49.684,159.140
C04803=1022.612,38.757,-102.652,167.220,49.688,159.140
C04804=1022.605,38.508,-102.636,167.217,49.693,159.141
C04805=1022.600,38.258,-102.621,167.214,49.698,159.141
C04806=1022.594,38.009,-102.605,167.212,49.702,159.142
C04807=1022.588,37.759,-102.588,167.209,49.707,159.142
C04808=1022.582,37.509,-102.573,167.207,49.712,159.143
C04809=1022.577,37.261,-102.557,167.204,49.716,159.143
C04810=1022.570,37.011,-102.542,167.202,49.720,159.144
C04811=1022.564,36.762,-102.526,167.199,49.725,159.144
C04812=1022.559,36.512,-102.510,167.196,49.729,159.144
C04813=1022.552,36.262,-102.495,167.194,49.734,159.145
C04814=1022.546,36.013,-102.479,167.191,49.739,159.145
C04815=1022.541,35.763,-102.464,167.188,49.744,159.146
C04816=1022.535,35.514,-102.448,167.186,49.748,159.146
C04817=1022.529,35.264,-102.433,167.183,49.753,159.147
C04818=1022.523,35.015,-102.418,167.181,49.757,159.147
C04819=1022.517,34.765,-102.401,167.178,49.762,159.148
C04820=1022.512,34.516,-102.386,167.175,49.767,159.148
C04821=1022.505,34.267,-102.371,167.173,49.772,159.149
C04822=1022.499,34.017,-102.355,167.170,49.776,159.149
C04823=1022.493,33.767,-102.340,167.168,49.780,159.149
C04824=1022.488,33.519,-102.324,167.164,49.785,159.150
C04825=1022.482,33.269,-102.309,167.162,49.790,159.150
C04826=1022.476,33.019,-102.294,167.160,49.795,159.151
C04827=1022.470,32.770,-102.277,167.157,49.799,159.151
C04828=1022.464,32.521,-102.263,167.155,49.804,159.152
C04829=1022.458,32.271,-102.247,167.151,49.809,159.152
C04830=1022.452,32.022,-102.232,167.149,49.813,159.153
C04831=1022.446,31.772,-102.216,167.146,49.817,159.153
C04832=1022.441,31.523,-102.201,167.144,49.822,159.154
C04833=1022.434,31.274,-102.185,167.142,49.827,159.154
C04834=1022.429,31.024,-102.170,167.138,49.831,159.154
C04835=1022.423,30.775,-102.155,167.136,49.836,159.155
C04836=1022.417,30.525,-102.139,167.133,49.841,159.155
C04837=1022.410,30.276,-102.124,167.131,49.845,159.156
C04838=1022.405,30.026,-102.108,167.128,49.849,159.156
C04839=1022.400,29.776,-102.093,167.125,49.854,159.157
C04840=1022.393,29.527,-102.078,167.123,49.859,159.157
C04841=1022.387,29.277,-102.062,167.120,49.863,159.157
C04842=1022.382,29.028,-102.047,167.118,49.868,159.158
C04843=1022.376,28.778,-102.032,167.115,49.873,159.158
C04844=1022.369,28.529,-102.016,167.113,49.877,159.159
C04845=1022.364,28.280,-102.001,167.109,49.882,159.159
C04846=1022.359,28.030,-101.986,167.107,49.886,159.160
C04847=1022.352,27.781,-101.971,167.104,49.890,159.160
C04848=1022.345,27.496,-101.953,167.101,49.896,159.161
C04849=1022.339,27.212,-101.936,167.098,49.901,159.161
C04850=1022.332,26.928,-101.919,167.095,49.906,159.161
C04851=1022.326,26.643,-101.901,167.093,49.912,159.162
C04852=1022.319,26.393,-101.886,167.089,49.917,159.163
C04853=1022.314,26.144,-101.872,167.087,49.921,159.163
C04854=1022.308,25.894,-101.856,167.085,49.926,159.163
C04855=1022.301,25.645,-101.840,167.082,49.930,159.164
C04856=1022.295,25.396,-101.826,167.080,49.935,159.165
C04857=1022.290,25.146,-101.810,167.076,49.939,159.165
C04858=1022.284,24.897,-101.796,167.074,49.944,159.165
C04859=1022.278,24.648,-101.781,167.072,49.949,159.166
C04860=1022.272,24.398,-101.765,167.069,49.954,159.166
C04861=1022.266,24.149,-101.751,167.066,49.958,159.166
C04862=1022.260,23.899,-101.736,167.063,49.963,159.167
C04863=1022.254,23.649,-101.720,167.061,49.967,159.168
C04864=1022.248,23.400,-101.706,167.058,49.971,159.168
C04865=1022.242,23.151,-101.691,167.055,49.976,159.168
C04866=1022.237,22.901,-101.675,167.053,49.981,159.169
C04867=1022.231,22.652,-101.660,167.050,49.986,159.169
C04868=1022.224,22.402,-101.646,167.048,49.990,159.170
C04869=1022.219,22.153,-101.630,167.044,49.995,159.170
C04870=1022.213,21.903,-101.615,167.042,50.000,159.171
C04871=1022.207,21.654,-101.601,167.039,50.004,159.171
C04872=1022.201,21.404,-101.585,167.037,50.009,159.171
C04873=1022.196,21.155,-101.571,167.035,50.013,159.172
C04874=1022.189,20.906,-101.556,167.031,50.018,159.172
C04875=1022.184,20.655,-101.541,167.029,50.022,159.173
C04876=1022.178,20.406,-101.526,167.027,50.027,159.173
C04877=1022.172,20.156,-101.511,167.024,50.031,159.173
C04878=1022.166,19.907,-101.497,167.021,50.036,159.174
C04879=1022.160,19.657,-101.481,167.018,50.041,159.174
C04880=1022.155,19.408,-101.467,167.016,50.045,159.175
C04881=1022.148,19.159,-101.452,167.013,50.050,159.175
C04882=1022.143,18.910,-101.437,167.011,50.055,159.176
C04883=1022.137,18.660,-101.422,167.007,50.059,159.176
C04884=1022.131,18.410,-101.408,167.005,50.064,159.177
C04885=1022.125,18.161,-101.393,167.003,50.068,159.177
C04886=1022.118,17.911,-101.378,166.999,50.073,159.177
C04887=1022.113,17.662,-101.363,166.997,50.078,159.178
C04888=1022.107,17.412,-101.348,166.994,50.082,159.178
C04889=1022.102,17.162,-101.334,166.992,50.086,159.179
C04890=1022.095,16.913,-101.319,166.988,50.091,159.179
C04891=1022.089,16.664,-101.304,166.986,50.096,159.180
C04892=1022.083,16.414,-101.289,166.984,50.101,159.180
C04893=1022.078,16.165,-101.276,166.981,50.105,159.180
C04894=1022.072,15.915,-101.260,166.978,50.110,159.181
C04895=1022.066,15.666,-101.245,166.975,50.114,159.181
C04896=1022.060,15.417,-101.231,166.973,50.119,159.182
C04897=1022.054,15.166,-101.217,166.971,50.124,159.182
C04898=1022.048,14.918,-101.202,166.968,50.128,159.182
C04899=1022.042,14.668,-101.187,166.965,50.133,159.183
C04900=1022.036,14.419,-101.173,166.962,50.138,159.183
C04901=1022.031,14.168,-101.158,166.960,50.142,159.184
C04902=1022.025,13.919,-101.143,166.957,50.146,159.184
C04903=1022.019,13.670,-101.128,166.954,50.151,159.185
C04904=1022.013,13.420,-101.114,166.952,50.156,159.185
C04905=1022.007,13.170,-101.099,166.949,50.160,159.185
C04906=1022.001,12.921,-101.086,166.946,50.165,159.186
C04907=1021.995,12.671,-101.071,166.943,50.169,159.186
C04908=1021.990,12.422,-101.057,166.941,50.174,159.187
C04909=1021.983,12.173,-101.043,166.938,50.179,159.187
C04910=1021.977,11.923,-101.028,166.935,50.184,159.188
C04911=1021.971,11.674,-101.014,166.933,50.189,159.188
C04912=1021.966,11.456,-101.001,166.930,50.193,159.188
C04913=1021.960,11.240,-100.989,166.928,50.197,159.189
C04914=1021.956,11.022,-100.976,166.926,50.201,159.189
C04915=1021.951,10.805,-100.964,166.924,50.205,159.189
C04916=1021.945,10.589,-100.951,166.921,50.209,159.190
C04917=1021.940,10.371,-100.939,166.918,50.213,159.190
C04918=1021.935,10.154,-100.926,166.917,50.217,159.191
C04919=1021.930,9.937,-100.914,166.914,50.221,159.191
C04920=1021.924,9.688,-100.900,166.911,50.226,159.191
C04921=1021.918,9.437,-100.885,166.908,50.231,159.192
C04922=1021.912,9.188,-100.871,166.906,50.235,159.192
C04923=1021.906,8.939,-100.858,166.903,50.239,159.193
C04924=1021.899,8.689,-100.843,166.900,50.244,159.193
C04925=1021.894,8.440,-100.829,166.898,50.249,159.194
C04926=1021.888,8.191,-100.814,166.895,50.253,159.194
C04927=1021.882,7.941,-100.800,166.892,50.258,159.194
C04928=1021.877,7.691,-100.786,166.890,50.263,159.195
C04929=1021.870,7.441,-100.771,166.887,50.268,159.195
C04930=1021.865,7.192,-100.757,166.884,50.272,159.196
C04931=1021.858,6.943,-100.743,166.881,50.277,159.196
C04932=1021.852,6.693,-100.729,166.879,50.281,159.196
C04933=1021.847,6.443,-100.715,166.877,50.286,159.197
C04934=1021.841,6.194,-100.701,166.873,50.291,159.197
C04935=1021.835,5.944,-100.686,166.871,50.295,159.198
C04936=1021.829,5.695,-100.672,166.868,50.300,159.198
C04937=1021.823,5.446,-100.658,166.865,50.305,159.198
C04938=1021.817,5.196,-100.644,166.862,50.309,159.199
C04939=1021.811,4.947,-100.630,166.860,50.314,159.199
C04940=1021.805,4.697,-100.616,166.857,50.319,159.200
C04941=1021.800,4.447,-100.602,166.854,50.323,159.200
C04942=1021.794,4.198,-100.587,166.852,50.328,159.201
C04943=1021.788,3.948,-100.573,166.849,50.332,159.201
C04944=1021.783,3.699,-100.559,166.846,50.337,159.201
C04945=1021.776,3.449,-100.546,166.843,50.341,159.202
C04946=1021.770,3.200,-100.531,166.841,50.346,159.202
C04947=1021.765,2.950,-100.517,166.839,50.351,159.203
C04948=1021.759,2.701,-100.503,166.835,50.355,159.203
C04949=1021.753,2.451,-100.488,166.833,50.360,159.203
C04950=1021.747,2.201,-100.475,166.830,50.364,159.204
C04951=1021.741,1.952,-100.461,166.827,50.369,159.204
C04952=1021.735,1.703,-100.447,166.824,50.373,159.204
C04953=1021.729,1.453,-100.433,166.822,50.378,159.205
C04954=1021.724,1.203,-100.419,166.819,50.382,159.205
C04955=1021.718,0.954,-100.405,166.816,50.387,159.206
C04956=1021.713,0.704,-100.391,166.814,50.392,159.206
C04957=1021.706,0.455,-100.377,166.811,50.396,159.206
C04958=1021.700,0.205,-100.363,166.809,50.401,159.207
C04959=1021.695,-0.044,-100.349,166.805,50.405,159.207
C04960=1021.689,-0.294,-100.335,166.803,50.410,159.208
C04961=1021.684,-0.543,-100.321,166.800,50.414,159.208
C04962=1021.677,-0.793,-100.306,166.797,50.419,159.208
C04963=1021.671,-1.042,-100.293,166.794,50.423,159.209
C04964=1021.666,-1.292,-100.279,166.792,50.427,159.209
C04965=1021.660,-1.542,-100.265,166.789,50.432,159.209
C04966=1021.655,-1.791,-100.251,166.786,50.436,159.210
C04967=1021.649,-2.041,-100.237,166.784,50.441,159.210
C04968=1021.643,-2.290,-100.223,166.781,50.445,159.211
C04969=1021.637,-2.540,-100.209,166.779,50.450,159.211
C04970=1021.631,-2.789,-100.195,166.775,50.455,159.211
C04971=1021.626,-3.039,-100.182,166.773,50.459,159.212
C04972=1021.618,-3.387,-100.162,166.769,50.466,159.212
C04973=1021.610,-3.735,-100.143,166.765,50.472,159.213
C04974=1021.602,-4.083,-100.123,166.761,50.478,159.213
C04975=1021.594,-4.430,-100.104,166.757,50.485,159.214
C04976=1021.587,-4.712,-100.089,166.754,50.490,159.214
C04977=1021.580,-4.993,-100.074,166.752,50.495,159.215
C04978=1021.573,-5.273,-100.058,166.749,50.500,159.215
C04979=1021.567,-5.555,-100.043,166.745,50.505,159.215
C04980=1021.561,-5.805,-100.030,166.742,50.510,159.216
C04981=1021.555,-6.054,-100.016,166.740,50.515,159.216
C04982=1021.549,-6.304,-100.002,166.737,50.519,159.217
C04983=1021.543,-6.553,-99.989,166.734,50.524,159.217
C04984=1021.537,-6.803,-99.975,166.732,50.529,159.218
C04985=1021.531,-7.052,-99.962,166.729,50.533,159.218
C04986=1021.525,-7.302,-99.949,166.726,50.538,159.218
C04987=1021.520,-7.552,-99.935,166.723,50.542,159.219
C04988=1021.513,-7.801,-99.922,166.720,50.547,159.219
C04989=1021.508,-8.051,-99.908,166.717,50.552,159.220
C04990=1021.502,-8.300,-99.895,166.715,50.556,159.220
C04991=1021.496,-8.549,-99.881,166.712,50.561,159.220
C04992=1021.490,-8.799,-99.868,166.709,50.565,159.221
C04993=1021.485,-9.049,-99.855,166.707,50.570,159.221
C04994=1021.479,-9.298,-99.841,166.703,50.575,159.221
C04995=1021.472,-9.548,-99.827,166.701,50.579,159.222
C04996=1021.466,-9.798,-99.814,166.699,50.584,159.222
C04997=1021.461,-10.048,-99.801,166.695,50.589,159.222
C04998=1021.455,-10.297,-99.787,166.693,50.593,159.223
C04999=1021.449,-10.546,-99.774,166.690,50.598,159.223
C05000=1021.443,-10.796,-99.760,166.687,50.603,159.224
C05001=1021.437,-11.045,-99.747,166.684,50.607,159.224
C05002=1021.432,-11.295,-99.734,166.682,50.612,159.224
C05003=1021.426,-11.545,-99.721,166.678,50.616,159.225
C05004=1021.420,-11.794,-99.707,166.676,50.621,159.225
C05005=1021.414,-12.044,-99.694,166.673,50.625,159.225
C05006=1021.409,-12.294,-99.680,166.670,50.630,159.226
C05007=1021.402,-12.543,-99.667,166.667,50.634,159.226
C05008=1021.396,-12.792,-99.654,166.665,50.639,159.227
C05009=1021.391,-13.042,-99.641,166.662,50.643,159.227
C05010=1021.385,-13.292,-99.627,166.659,50.648,159.227
C05011=1021.379,-13.541,-99.613,166.657,50.652,159.228
C05012=1021.374,-13.791,-99.601,166.653,50.657,159.228
C05013=1021.368,-14.041,-99.587,166.651,50.662,159.228
C05014=1021.362,-14.290,-99.574,166.648,50.666,159.229
C05015=1021.357,-14.540,-99.561,166.645,50.671,159.229
C05016=1021.350,-14.790,-99.547,166.642,50.675,159.229
C05017=1021.344,-15.039,-99.534,166.640,50.680,159.230
C05018=1021.339,-15.289,-99.521,166.636,50.684,159.230
C05019=1021.333,-15.538,-99.508,166.634,50.688,159.230
C05020=1021.327,-15.788,-99.494,166.632,50.693,159.231
C05021=1021.322,-16.037,-99.482,166.628,50.698,159.231
C05022=1021.316,-16.286,-99.468,166.626,50.702,159.232
C05023=1021.310,-16.536,-99.456,166.623,50.707,159.232
C05024=1021.304,-16.786,-99.442,166.620,50.712,159.232
C05025=1021.299,-17.036,-99.429,166.618,50.717,159.233
C05026=1021.292,-17.285,-99.416,166.614,50.721,159.233
C05027=1021.286,-17.535,-99.404,166.612,50.726,159.234
C05028=1021.280,-17.784,-99.390,166.609,50.730,159.234
C05029=1021.274,-18.034,-99.378,166.606,50.735,159.234
C05030=1021.269,-18.284,-99.365,166.604,50.740,159.235
C05031=1021.263,-18.533,-99.351,166.600,50.744,159.235
C05032=1021.257,-18.783,-99.339,166.598,50.749,159.235
C05033=1021.251,-19.032,-99.325,166.595,50.753,159.236
C05034=1021.245,-19.282,-99.313,166.592,50.758,159.236
C05035=1021.239,-19.531,-99.300,166.589,50.763,159.236
C05036=1021.234,-19.781,-99.287,166.586,50.768,159.237
C05037=1021.228,-20.031,-99.274,166.583,50.772,159.237
C05038=1021.222,-20.280,-99.261,166.581,50.777,159.238
C05039=1021.216,-20.530,-99.248,166.577,50.781,159.238
C05040=1021.210,-20.810,-99.234,166.574,50.786,159.238
C05041=1021.203,-21.089,-99.220,166.571,50.791,159.239
C05042=1021.197,-21.368,-99.205,166.568,50.797,159.239
C05043=1021.190,-21.648,-99.191,166.565,50.801,159.239
C05044=1021.184,-21.897,-99.178,166.562,50.807,159.240
C05045=1021.179,-22.146,-99.165,166.560,50.811,159.240
C05046=1021.173,-22.396,-99.153,166.556,50.816,159.241
C05047=1021.167,-22.645,-99.140,166.554,50.820,159.241
C05048=1021.161,-22.895,-99.126,166.551,50.825,159.241
C05049=1021.155,-23.145,-99.114,166.548,50.829,159.242
C05050=1021.149,-23.395,-99.101,166.545,50.833,159.242
C05051=1021.144,-23.644,-99.088,166.542,50.839,159.242
C05052=1021.138,-23.894,-99.076,166.539,50.843,159.243
C05053=1021.132,-24.144,-99.063,166.537,50.848,159.243
C05054=1021.126,-24.393,-99.050,166.533,50.852,159.243
C05055=1021.121,-24.642,-99.037,166.531,50.857,159.244
C05056=1021.115,-24.892,-99.025,166.529,50.861,159.244
C05057=1021.110,-25.142,-99.012,166.525,50.865,159.244
C05058=1021.103,-25.391,-98.999,166.523,50.870,159.245
C05059=1021.097,-25.641,-98.986,166.520,50.874,159.245
C05060=1021.092,-25.890,-98.974,166.517,50.880,159.245
C05061=1021.086,-26.140,-98.962,166.514,50.884,159.246
C05062=1021.080,-26.390,-98.948,166.511,50.888,159.246
C05063=1021.075,-26.640,-98.935,166.508,50.893,159.246
C05064=1021.070,-26.889,-98.923,166.506,50.897,159.247
C05065=1021.064,-27.139,-98.910,166.502,50.902,159.247
C05066=1021.058,-27.389,-98.898,166.500,50.907,159.247
C05067=1021.052,-27.639,-98.885,166.497,50.911,159.248
C05068=1021.046,-27.888,-98.873,166.494,50.916,159.248
C05069=1021.040,-28.137,-98.860,166.492,50.920,159.248
C05070=1021.034,-28.387,-98.847,166.488,50.925,159.249
C05071=1021.028,-28.637,-98.835,166.486,50.929,159.249
C05072=1021.023,-28.886,-98.823,166.482,50.934,159.249
C05073=1021.016,-29.136,-98.811,166.480,50.939,159.250
C05074=1021.011,-29.385,-98.798,166.477,50.944,159.250
C05075=1021.005,-29.635,-98.786,166.474,50.948,159.250
C05076=1020.999,-29.884,-98.773,166.472,50.953,159.251
C05077=1020.993,-30.134,-98.761,166.468,50.957,159.251
C05078=1020.988,-30.384,-98.748,166.466,50.962,159.252
C05079=1020.982,-30.633,-98.736,166.462,50.967,159.252
C05080=1020.976,-30.883,-98.724,166.460,50.971,159.252
C05081=1020.970,-31.133,-98.711,166.456,50.976,159.252
C05082=1020.964,-31.382,-98.699,166.454,50.981,159.253
C05083=1020.958,-31.632,-98.687,166.451,50.985,159.253
C05084=1020.953,-31.882,-98.675,166.448,50.989,159.253
C05085=1020.948,-32.132,-98.663,166.446,50.994,159.254
C05086=1020.942,-32.382,-98.650,166.442,50.999,159.254
C05087=1020.936,-32.630,-98.639,166.440,51.004,159.255
C05088=1020.930,-32.880,-98.626,166.436,51.008,159.255
C05089=1020.924,-33.130,-98.613,166.434,51.013,159.255
C05090=1020.918,-33.379,-98.601,166.430,51.017,159.255
C05091=1020.913,-33.629,-98.589,166.428,51.022,159.256
C05092=1020.907,-33.879,-98.576,166.426,51.026,159.256
C05093=1020.901,-34.128,-98.565,166.422,51.031,159.256
C05094=1020.895,-34.378,-98.552,166.420,51.036,159.257
C05095=1020.890,-34.628,-98.541,166.416,51.040,159.257
C05096=1020.884,-34.878,-98.528,166.414,51.044,159.257
C05097=1020.878,-35.127,-98.515,166.410,51.050,159.258
C05098=1020.873,-35.377,-98.503,166.408,51.054,159.258
C05099=1020.866,-35.626,-98.491,166.405,51.058,159.258
C05100=1020.861,-35.875,-98.479,166.402,51.063,159.259
C05101=1020.855,-36.126,-98.467,166.399,51.067,159.259
C05102=1020.850,-36.375,-98.455,166.396,51.072,159.259
C05103=1020.844,-36.625,-98.443,166.394,51.077,159.260
C05104=1020.837,-36.903,-98.429,166.390,51.082,159.260
C05105=1020.831,-37.182,-98.416,166.387,51.087,159.260
C05106=1020.825,-37.460,-98.402,166.383,51.091,159.261
C05107=1020.818,-37.739,-98.388,166.380,51.097,159.261
C05108=1020.813,-37.988,-98.377,166.378,51.101,159.261
C05109=1020.807,-38.238,-98.364,166.375,51.106,159.262
C05110=1020.801,-38.487,-98.353,166.372,51.110,159.262
C05111=1020.795,-38.737,-98.340,166.369,51.114,159.262
C05112=1020.790,-38.987,-98.328,166.366,51.120,159.263
C05113=1020.784,-39.237,-98.316,166.363,51.124,159.263
C05114=1020.778,-39.487,-98.303,166.360,51.128,159.263
C05115=1020.773,-39.736,-98.293,166.358,51.133,159.264
C05116=1020.767,-39.986,-98.280,166.354,51.138,159.264
C05117=1020.761,-40.235,-98.269,166.352,51.142,159.264
C05118=1020.755,-40.485,-98.257,166.348,51.147,159.264
C05119=1020.749,-40.734,-98.245,166.346,51.152,159.265
C05120=1020.744,-40.984,-98.233,166.343,51.156,159.265
C05121=1020.738,-41.234,-98.221,166.340,51.161,159.266
C05122=1020.732,-41.483,-98.210,166.337,51.165,159.266
C05123=1020.727,-41.733,-98.197,166.334,51.170,159.266
C05124=1020.721,-41.983,-98.187,166.332,51.175,159.267
C05125=1020.715,-42.233,-98.174,166.328,51.179,159.267
C05126=1020.709,-42.482,-98.163,166.326,51.184,159.267
C05127=1020.703,-42.732,-98.151,166.322,51.189,159.267
C05128=1020.698,-42.982,-98.140,166.320,51.193,159.268
C05129=1020.692,-43.231,-98.127,166.316,51.198,159.268
C05130=1020.687,-43.481,-98.116,166.314,51.202,159.268
C05131=1020.681,-43.730,-98.104,166.311,51.207,159.269
C05132=1020.675,-43.981,-98.092,166.308,51.211,159.269
C05133=1020.669,-44.229,-98.081,166.304,51.216,159.269
C05134=1020.663,-44.480,-98.069,166.302,51.221,159.270
C05135=1020.657,-44.729,-98.057,166.299,51.225,159.270
C05136=1020.652,-44.979,-98.045,166.296,51.230,159.270
C05137=1020.646,-45.228,-98.034,166.293,51.235,159.271
C05138=1020.641,-45.478,-98.022,166.290,51.239,159.271
C05139=1020.634,-45.728,-98.010,166.288,51.243,159.271
C05140=1020.629,-45.977,-97.999,166.284,51.248,159.271
C05141=1020.624,-46.227,-97.987,166.282,51.252,159.272
C05142=1020.617,-46.477,-97.975,166.278,51.257,159.272
C05143=1020.612,-46.727,-97.964,166.276,51.262,159.272
C05144=1020.606,-46.975,-97.952,166.272,51.266,159.273
C05145=1020.601,-47.226,-97.941,166.270,51.271,159.273
C05146=1020.595,-47.475,-97.930,166.267,51.276,159.273
C05147=1020.589,-47.725,-97.917,166.264,51.280,159.274
C05148=1020.583,-47.975,-97.906,166.260,51.284,159.274
C05149=1020.578,-48.225,-97.895,166.258,51.289,159.274
C05150=1020.572,-48.473,-97.883,166.256,51.294,159.275
C05151=1020.567,-48.724,-97.871,166.252,51.298,159.275
C05152=1020.561,-48.973,-97.860,166.249,51.302,159.275
C05153=1020.556,-49.223,-97.848,166.246,51.307,159.275
C05154=1020.550,-49.473,-97.836,166.244,51.312,159.276
C05155=1020.544,-49.723,-97.826,166.240,51.316,159.276
C05156=1020.539,-49.972,-97.813,166.237,51.320,159.276
C05157=1020.533,-50.222,-97.802,166.234,51.326,159.276
C05158=1020.528,-50.472,-97.791,166.232,51.330,159.277
C05159=1020.522,-50.721,-97.779,166.229,51.334,159.277
C05160=1020.517,-50.970,-97.768,166.225,51.338,159.277
C05161=1020.510,-51.221,-97.756,166.223,51.343,159.278
C05162=1020.504,-51.470,-97.746,166.220,51.348,159.278
C05163=1020.499,-51.720,-97.735,166.216,51.353,159.278
C05164=1020.492,-51.970,-97.723,166.214,51.357,159.278
C05165=1020.487,-52.219,-97.713,166.211,51.362,159.279
C05166=1020.481,-52.469,-97.702,166.208,51.367,159.279
C05167=1020.476,-52.719,-97.690,166.205,51.372,159.280
C05168=1020.469,-52.997,-97.678,166.202,51.377,159.280
C05169=1020.463,-53.276,-97.665,166.198,51.382,159.280
C05170=1020.456,-53.555,-97.653,166.195,51.388,159.281
C05171=1020.449,-53.834,-97.640,166.192,51.393,159.281
C05172=1020.444,-54.083,-97.630,166.188,51.397,159.281
C05173=1020.438,-54.333,-97.619,166.186,51.402,159.282
C05174=1020.432,-54.582,-97.608,166.183,51.407,159.282
C05175=1020.426,-54.833,-97.596,166.179,51.412,159.282
C05176=1020.421,-55.082,-97.585,166.177,51.416,159.282
C05177=1020.415,-55.332,-97.574,166.173,51.421,159.283
C05178=1020.409,-55.581,-97.563,166.171,51.426,159.283
C05179=1020.403,-55.831,-97.552,166.167,51.430,159.283
C05180=1020.397,-56.081,-97.541,166.165,51.435,159.284
C05181=1020.391,-56.330,-97.530,166.162,51.440,159.284
C05182=1020.386,-56.580,-97.519,166.159,51.444,159.284
C05183=1020.380,-56.829,-97.509,166.156,51.449,159.285
C05184=1020.375,-57.080,-97.498,166.152,51.454,159.285
C05185=1020.369,-57.329,-97.487,166.150,51.458,159.285
///RCONF 1,0,0,1,0,0,0,0,0,0,0,0,0,0,0,0,0,0,0,0,0,0,0,0
C05186=1020.363,-57.580,-97.476,166.146,51.463,159.285
C05187=1020.357,-57.829,-97.465,166.144,51.467,159.286
C05188=1020.352,-58.079,-97.454,166.141,51.472,159.286
C05189=1020.346,-58.328,-97.443,166.138,51.477,159.286
C05190=1020.340,-58.577,-97.432,166.135,51.481,159.286
C05191=1020.334,-58.827,-97.421,166.132,51.486,159.287
C05192=1020.329,-59.077,-97.410,166.129,51.491,159.287
C05193=1020.323,-59.328,-97.399,166.127,51.496,159.288
C05194=1020.318,-59.577,-97.388,166.123,51.500,159.288
C05195=1020.312,-59.827,-97.378,166.119,51.505,159.288
C05196=1020.306,-60.076,-97.367,166.117,51.509,159.288
C05197=1020.300,-60.326,-97.356,166.114,51.514,159.289
C05198=1020.295,-60.575,-97.345,166.111,51.518,159.289
C05199=1020.289,-60.825,-97.335,166.107,51.523,159.289
C05200=1020.284,-61.075,-97.324,166.105,51.528,159.289
C05201=1020.278,-61.324,-97.313,166.102,51.532,159.290
C05202=1020.273,-61.574,-97.302,166.099,51.536,159.290
C05203=1020.267,-61.823,-97.291,166.096,51.542,159.290
C05204=1020.262,-62.074,-97.280,166.093,51.546,159.291
C05205=1020.256,-62.323,-97.270,166.090,51.550,159.291
C05206=1020.250,-62.573,-97.259,166.087,51.555,159.291
C05207=1020.244,-62.823,-97.247,166.084,51.560,159.291
C05208=1020.238,-63.073,-97.237,166.081,51.564,159.292
C05209=1020.233,-63.322,-97.226,166.078,51.569,159.292
C05210=1020.227,-63.572,-97.216,166.076,51.574,159.292
C05211=1020.221,-63.822,-97.205,166.072,51.578,159.292
C05212=1020.216,-64.071,-97.195,166.069,51.582,159.293
C05213=1020.211,-64.321,-97.183,166.066,51.587,159.293
C05214=1020.205,-64.571,-97.172,166.063,51.591,159.293
C05215=1020.200,-64.821,-97.162,166.060,51.596,159.293
C05216=1020.194,-65.070,-97.151,166.058,51.601,159.294
C05217=1020.188,-65.320,-97.140,166.054,51.605,159.294
C05218=1020.183,-65.570,-97.130,166.051,51.609,159.294
C05219=1020.177,-65.819,-97.120,166.048,51.615,159.295
C05220=1020.172,-66.068,-97.109,166.046,51.619,159.295
C05221=1020.166,-66.318,-97.099,166.042,51.623,159.295
C05222=1020.161,-66.568,-97.088,166.040,51.627,159.295
C05223=1020.155,-66.818,-97.078,166.036,51.632,159.295
C05224=1020.149,-67.067,-97.067,166.033,51.636,159.296
C05225=1020.144,-67.317,-97.055,166.030,51.642,159.296
C05226=1020.139,-67.567,-97.045,166.028,51.646,159.296
C05227=1020.133,-67.817,-97.034,166.024,51.650,159.296
C05228=1020.128,-68.067,-97.024,166.021,51.654,159.297
C05229=1020.122,-68.316,-97.013,166.018,51.659,159.297
C05230=1020.116,-68.566,-97.002,166.015,51.663,159.297
C05231=1020.111,-68.816,-96.992,166.012,51.669,159.298
C05232=1020.105,-69.096,-96.980,166.009,51.673,159.298
C05233=1020.099,-69.376,-96.969,166.005,51.678,159.298
C05234=1020.093,-69.655,-96.957,166.002,51.683,159.298
C05235=1020.086,-69.935,-96.945,165.999,51.688,159.299
C05236=1020.080,-70.185,-96.935,165.996,51.692,159.299
C05237=1020.076,-70.435,-96.924,165.992,51.697,159.299
C05238=1020.071,-70.685,-96.913,165.990,51.701,159.299
C05239=1020.065,-70.934,-96.903,165.987,51.705,159.300
C05240=1020.059,-71.184,-96.892,165.984,51.711,159.300
C05241=1020.054,-71.434,-96.882,165.982,51.715,159.300
C05242=1020.048,-71.684,-96.871,165.978,51.719,159.300
C05243=1020.043,-71.933,-96.861,165.975,51.724,159.301
C05244=1020.038,-72.183,-96.851,165.972,51.728,159.301
C05245=1020.032,-72.432,-96.840,165.969,51.732,159.301
C05246=1020.027,-72.682,-96.830,165.966,51.737,159.301
C05247=1020.021,-72.932,-96.819,165.963,51.741,159.301
C05248=1020.016,-73.181,-96.809,165.961,51.745,159.302
C05249=1020.011,-73.431,-96.799,165.957,51.750,159.302
C05250=1020.005,-73.681,-96.788,165.954,51.754,159.302
C05251=1019.999,-73.931,-96.778,165.951,51.759,159.302
C05252=1019.994,-74.180,-96.767,165.948,51.763,159.303
C05253=1019.989,-74.430,-96.757,165.945,51.768,159.303
C05254=1019.983,-74.680,-96.747,165.942,51.772,159.303
C05255=1019.978,-74.930,-96.737,165.939,51.777,159.303
C05256=1019.972,-75.180,-96.726,165.936,51.781,159.304
C05257=1019.966,-75.429,-96.716,165.933,51.786,159.304
C05258=1019.961,-75.679,-96.707,165.930,51.790,159.304
C05259=1019.956,-75.929,-96.696,165.927,51.795,159.304
C05260=1019.950,-76.179,-96.686,165.925,51.800,159.305
C05261=1019.944,-76.428,-96.676,165.921,51.804,159.305
C05262=1019.939,-76.678,-96.666,165.917,51.809,159.305
C05263=1019.934,-76.928,-96.656,165.915,51.813,159.305
C05264=1019.928,-77.178,-96.646,165.912,51.818,159.306
C05265=1019.922,-77.428,-96.636,165.909,51.823,159.306
C05266=1019.917,-77.676,-96.626,165.905,51.827,159.306
C05267=1019.911,-77.927,-96.616,165.903,51.831,159.306
C05268=1019.906,-78.177,-96.605,165.899,51.836,159.306
C05269=1019.900,-78.426,-96.596,165.897,51.840,159.307
C05270=1019.895,-78.676,-96.586,165.894,51.845,159.307
C05271=1019.890,-78.926,-96.576,165.891,51.850,159.307
C05272=1019.885,-79.175,-96.566,165.887,51.854,159.307
C05273=1019.879,-79.425,-96.557,165.885,51.858,159.308
C05274=1019.873,-79.675,-96.546,165.881,51.863,159.308
C05275=1019.868,-79.924,-96.536,165.879,51.867,159.308
C05276=1019.863,-80.174,-96.526,165.875,51.872,159.308
C05277=1019.856,-80.424,-96.516,165.873,51.877,159.309
C05278=1019.852,-80.673,-96.506,165.870,51.881,159.309
C05279=1019.845,-80.923,-96.497,165.866,51.886,159.309
C05280=1019.840,-81.174,-96.487,165.864,51.891,159.310
C05281=1019.835,-81.423,-96.478,165.860,51.895,159.310
C05282=1019.829,-81.673,-96.468,165.858,51.900,159.310
C05283=1019.823,-81.923,-96.458,165.854,51.905,159.310
C05284=1019.817,-82.172,-96.449,165.851,51.910,159.310
C05285=1019.812,-82.422,-96.439,165.848,51.914,159.311
C05286=1019.806,-82.672,-96.430,165.845,51.918,159.311
C05287=1019.801,-82.921,-96.420,165.843,51.923,159.311
C05288=1019.795,-83.171,-96.410,165.839,51.928,159.311
C05289=1019.790,-83.421,-96.400,165.835,51.933,159.312
C05290=1019.784,-83.671,-96.391,165.833,51.938,159.312
C05291=1019.779,-83.921,-96.381,165.830,51.942,159.312
C05292=1019.773,-84.170,-96.372,165.827,51.946,159.312
C05293=1019.768,-84.420,-96.362,165.824,51.951,159.313
C05294=1019.762,-84.669,-96.353,165.821,51.955,159.313
C05295=1019.757,-84.919,-96.343,165.818,51.960,159.313
C05296=1019.750,-85.201,-96.333,165.815,51.966,159.314
C05297=1019.744,-85.484,-96.322,165.811,51.970,159.314
C05298=1019.738,-85.765,-96.311,165.807,51.976,159.314
C05299=1019.732,-86.047,-96.300,165.804,51.981,159.314
C05300=1019.726,-86.297,-96.291,165.801,51.986,159.315
C05301=1019.721,-86.547,-96.281,165.798,51.990,159.315
C05302=1019.715,-86.796,-96.272,165.795,51.994,159.315
C05303=1019.710,-87.046,-96.262,165.792,52.000,159.315
C05304=1019.704,-87.296,-96.253,165.789,52.004,159.316
C05305=1019.699,-87.546,-96.243,165.786,52.009,159.316
C05306=1019.693,-87.795,-96.234,165.782,52.013,159.316
C05307=1019.688,-88.045,-96.225,165.780,52.017,159.316
C05308=1019.683,-88.295,-96.215,165.776,52.022,159.316
C05309=1019.677,-88.544,-96.206,165.774,52.027,159.317
C05310=1019.672,-88.794,-96.196,165.771,52.032,159.317
C05311=1019.666,-89.044,-96.187,165.768,52.036,159.317
C05312=1019.661,-89.294,-96.177,165.764,52.040,159.317
C05313=1019.655,-89.543,-96.168,165.762,52.045,159.317
C05314=1019.650,-89.794,-96.158,165.758,52.049,159.318
C05315=1019.645,-90.043,-96.149,165.756,52.054,159.318
C05316=1019.638,-90.293,-96.139,165.753,52.059,159.318
C05317=1019.634,-90.543,-96.130,165.749,52.063,159.318
C05318=1019.628,-90.792,-96.121,165.746,52.068,159.319
C05319=1019.623,-91.043,-96.112,165.743,52.072,159.319
C05320=1019.618,-91.292,-96.103,165.740,52.077,159.319
C05321=1019.612,-91.542,-96.092,165.737,52.081,159.319
C05322=1019.607,-91.792,-96.084,165.734,52.085,159.319
C05323=1019.601,-92.042,-96.074,165.731,52.090,159.320
C05324=1019.596,-92.292,-96.065,165.728,52.094,159.320
C05325=1019.591,-92.541,-96.056,165.725,52.100,159.320
C05326=1019.585,-92.791,-96.046,165.722,52.104,159.320
C05327=1019.580,-93.040,-96.037,165.719,52.108,159.321
C05328=1019.575,-93.290,-96.028,165.716,52.113,159.321
C05329=1019.569,-93.540,-96.019,165.713,52.117,159.321
C05330=1019.564,-93.789,-96.010,165.710,52.122,159.321
C05331=1019.559,-94.040,-96.000,165.707,52.126,159.321
C05332=1019.553,-94.289,-95.991,165.704,52.130,159.322
C05333=1019.548,-94.539,-95.982,165.701,52.135,159.322
C05334=1019.542,-94.789,-95.972,165.698,52.139,159.322
C05335=1019.537,-95.039,-95.964,165.695,52.144,159.322
C05336=1019.532,-95.288,-95.954,165.692,52.148,159.322
C05337=1019.526,-95.539,-95.945,165.688,52.153,159.322
C05338=1019.521,-95.788,-95.935,165.686,52.157,159.323
C05339=1019.516,-96.038,-95.927,165.682,52.162,159.323
C05340=1019.511,-96.287,-95.918,165.680,52.166,159.323
C05341=1019.505,-96.538,-95.908,165.676,52.171,159.323
C05342=1019.500,-96.787,-95.899,165.674,52.175,159.324
C05343=1019.495,-97.037,-95.890,165.670,52.179,159.324
C05344=1019.490,-97.287,-95.881,165.668,52.184,159.324
C05345=1019.485,-97.536,-95.871,165.665,52.188,159.324
C05346=1019.479,-97.786,-95.863,165.662,52.193,159.324
C05347=1019.473,-98.036,-95.853,165.659,52.197,159.325
C05348=1019.468,-98.286,-95.845,165.655,52.201,159.325
C05349=1019.463,-98.535,-95.836,165.652,52.207,159.325
C05350=1019.458,-98.785,-95.827,165.650,52.211,159.325
C05351=1019.452,-99.035,-95.818,165.646,52.216,159.325
C05352=1019.447,-99.285,-95.809,165.644,52.220,159.326
C05353=1019.442,-99.535,-95.801,165.640,52.225,159.326
C05354=1019.436,-99.784,-95.792,165.638,52.229,159.326
C05355=1019.430,-100.034,-95.783,165.634,52.233,159.326
C05356=1019.425,-100.284,-95.774,165.631,52.239,159.327
C05357=1019.420,-100.534,-95.765,165.628,52.243,159.327
C05358=1019.415,-100.784,-95.757,165.625,52.248,159.327
C05359=1019.409,-101.034,-95.748,165.622,52.252,159.327
C05360=1019.403,-101.318,-95.738,165.619,52.257,159.328
C05361=1019.397,-101.601,-95.728,165.614,52.262,159.327
C05362=1019.391,-101.885,-95.718,165.611,52.268,159.328
C05363=1019.385,-102.170,-95.708,165.608,52.273,159.328
C05364=1019.379,-102.419,-95.699,165.606,52.277,159.328
C05365=1019.374,-102.669,-95.690,165.602,52.282,159.329
C05366=1019.369,-102.919,-95.681,165.600,52.286,159.329
C05367=1019.364,-103.169,-95.673,165.596,52.291,159.329
C05368=1019.359,-103.419,-95.664,165.593,52.295,159.329
C05369=1019.353,-103.668,-95.656,165.590,52.300,159.329
C05370=1019.347,-103.919,-95.647,165.586,52.304,159.329
C05371=1019.342,-104.168,-95.639,165.584,52.309,159.330
C05372=1019.337,-104.418,-95.630,165.580,52.313,159.330
C05373=1019.331,-104.667,-95.621,165.578,52.317,159.330
C05374=1019.326,-104.917,-95.612,165.575,52.323,159.330
C05375=1019.321,-105.167,-95.604,165.572,52.327,159.331
C05376=1019.316,-105.417,-95.595,165.569,52.332,159.331
C05377=1019.311,-105.666,-95.586,165.566,52.336,159.331
C05378=1019.306,-105.916,-95.578,165.562,52.341,159.331
C05379=1019.300,-106.166,-95.569,165.560,52.345,159.331
C05380=1019.295,-106.416,-95.560,165.556,52.350,159.332
C05381=1019.289,-106.666,-95.552,165.554,52.354,159.332
C05382=1019.284,-106.916,-95.544,165.550,52.358,159.332
C05383=1019.279,-107.165,-95.535,165.548,52.363,159.332
C05384=1019.274,-107.415,-95.527,165.544,52.367,159.332
C05385=1019.268,-107.665,-95.518,165.542,52.372,159.333
C05386=1019.263,-107.914,-95.510,165.538,52.376,159.333
C05387=1019.258,-108.165,-95.502,165.536,52.381,159.333
C05388=1019.253,-108.415,-95.493,165.532,52.385,159.333
C05389=1019.248,-108.664,-95.485,165.530,52.390,159.333
